	2: (* === Check loop *)
		IF NOT (MB_Lock OR MB_Start) THEN
			WHILE VarCnt<=(VARS_Max-1) AND VarSta=2 DO
				(* Check only active vars *)
				IF VARS[VarCnt].Variable<>0 THEN			(* "Variable" is a pointer to word, so if 0 no address *)
					(* Check var auto-refresh on timer checks *)
					IF VARS[VarCnt].Refresh_Time>0 AND VARS[VarCnt].Refresh_Cnt=0 THEN
						VARS[VarCnt].Refresh_Cnt:=VARS[VarCnt].Refresh_Time;
						VarSta:=3;
					END_IF
					(* Check refresh for change or request *)
					CASE VARS[VarCnt].FunCode OF
						5,6,15,16: (* Write functions *)
							IF VARS[VarCnt].Variable_Size=1 THEN
								IF VARS[VarCnt].Variable^<>VARS[VarCnt].Variable_Mirror THEN
									VARS[VarCnt].Variable_Mirror:=VARS[VarCnt].Variable^;
									VarSta:=3;
								END_IF
							ELSE
								IF VARS[VarCnt].Variable_Mirror<>0 THEN
									VARS[VarCnt].Variable_Mirror:=0;
									VarSta:=3;
								END_IF
							END_IF
						1,2,3,4: (* Read functions *)
							IF VARS[VarCnt].Variable_Mirror<>0 THEN
								VARS[VarCnt].Variable_Mirror:=0;
								VarSta:=3;
							END_IF
					END_CASE
				END_IF
				(* Process query *)
				IF VarSta=3 THEN
					MB_Lock:=TRUE;
					MB_Query.SlaveAddress:=VARS[VarCnt].SlaveAddress;
					MB_Query.FunctionCode:=VARS[VarCnt].FunCode;
					CASE VARS[VarCnt].FunCode OF
						16#5,16#6,16#F,16#10:
							MB_Query.Read_Quantity:=0;
							MB_Query.Read_StartAddress:=0;
							MB_Query.Write_StartAddress:=VARS[VarCnt].FunAddress;
							MB_Query.Write_Quantity:=VARS[VarCnt].Variable_Size;
							IF VARS[VarCnt].Variable_Size=200 THEN
								COPY_32SWAP16(VARS[VarCnt].Variable, ADR(MB_Query.Write_Data[0]));
							ELSIF VARS[VarCnt].Variable_Size>1 THEN
								MEMCPY(VARS[VarCnt].Variable, ADR(MB_Query.Write_Data[0]), 2*VARS[VarCnt].Variable_Size);
							ELSE
								MB_Query.Write_Data[0]:=VARS[VarCnt].Variable^;
							END_IF
						16#1,16#2,16#3,16#4:
							MB_Query.Read_StartAddress:=VARS[VarCnt].FunAddress;
							IF VARS[VarCnt].Variable_Size=200 THEN MB_Query.Read_Quantity:=2; ELSE
							  MB_Query.Read_Quantity:=VARS[VarCnt].Variable_Size;
							END_IF
							MB_Query.Write_StartAddress:=0;
							MB_Query.Write_Quantity:=0;
					END_CASE
					VarRetry:=0;
					MB_Start:=TRUE;
				ELSE
					VarCnt:=VarCnt+1;
				END_IF
			END_WHILE
			(* Check loop completed -> no actions *)
			IF VarSta=2 THEN VarSta:=1; END_IF
		END_IF

	3: (* === Wait & process MB response *)
		IF NOT MB_Start THEN
			IF MB_MASTER.MB_Error=0 THEN
				CASE VARS[VarCnt].FunCode OF
					1,2,3,4:
						IF VARS[VarCnt].Variable_Size=200 THEN
							COPY_32SWAP16(ADR(MB_Resp.Data), VARS[VarCnt].Variable);
						ELSIF VARS[VarCnt].Variable_Size>1 THEN
							MEMCPY(ADR(MB_Resp.Data), VARS[VarCnt].Variable, 2*VARS[VarCnt].Variable_Size);
						ELSE
							VARS[VarCnt].Variable^:=MB_Resp.Data[0];
						END_IF
				END_CASE
				MB_Lock:=FALSE;
				(* Signal error recovery *)
				IF VARS_Alarm=TRUE AND VarCnt=VarAlarm THEN
					LogEv(EL_Wrn,EO_MODBUS,ID,5,'');
					VARS_Alarm:=FALSE;
				END_IF
				(* Next var *)
				VarCnt:=VarCnt+1;
				VarSta:=2;
			ELSE
				IF VarRetry<3 THEN
					VarRetry:=VarRetry+1;
					MB_Start:=TRUE;
				ELSE
					MB_Lock:=FALSE;
					(* Signal error *)
					IF VARS_Alarm=FALSE THEN
						LogEv(EL_Wrn,EO_MODBUS,ID,3,INT_TO_STRING(MB_MASTER.MB_Error));
						VARS_Alarm:=TRUE;
						VarAlarm:=VarCnt-1;
					END_IF
					(* Next var *)
					VarCnt:=VarCnt+1;
					VarSta:=2;
				END_IF
			END_IF
		END_IF

ELSE
	VarSta:=0;
END_CASE
END_ACTION

(* POU Plant_Objects/obj_MODBUS_CIR, ST *)
FUNCTION_BLOCK obj_MODBUS_CIR
VAR CONSTANT
	WAIT_STATE		:	BYTE := 0;
	PUMP_STATUS		:	BYTE := 1;
	PUMP_DATA		:	BYTE := 2;
	PUMP_ALARMS		:	BYTE := 3;
	PUMP_END_READ	:	BYTE := 4;
	CIR_ON_OFF		:	BYTE := 90;
	CIR_ON_OFF_CHECK:	BYTE := 91;
	CIR_END_WRITE	:	BYTE := 92;
	ERROR_STATE		:	BYTE := 100;
END_VAR
VAR_INPUT
	ID		:	BYTE;
	Address :	BYTE;		(* Pump address *)

	(* Physical inputs *)
	CIR_RUN_REQ		: BOOL; (* External run request (no heat or cold requested) *)
	CIR_STOP_REQ	: BOOL; (* External stop request (has priority over RUN signals!) *)

	Pump_AL			: BOOL; (* Alarm input signal *)
	Pump_AUTO		: BOOL;	(* Automatic/Manual input *)

	(* Controls *)
	OnOff		: 	BOOL;
	InitOK		:	BOOL;

	(* Timings *)
	OnDelay		:	TIME;
	OffDelay	:	TIME;

	(* Modbus *)
	Refresh_Now	:	BOOL;	(* Start immediately modbus state machine *)
END_VAR
VAR_IN_OUT
	ModBus		:	obj_MODBUS;
END_VAR
VAR_OUTPUT
	Ctrl_Run	:	BOOL;		(* Logical status of the device: 0: Not running (switched off), 1: running *)
	Run			:	BOOL;		(* Real status *)

	Status_Log	:	WORD;
	Status_Vis	:	DWORD;
END_VAR
VAR
	Pump_En		:	BOOL;

	(* Filters *)
	fPump_AL	:	FLT_EVENT := (INITEV:=FALSE);
	fPump_ST	:	FLT_EVENT := (INITEV:=FALSE);
	fPump_En	:	FLT_EVENT;
	fCIR_AUTO	:	FLT_EVENT;
	fStatus		:	FLT_EVENT;
	fStatusFault:	BOOL;

	(* Timer manage switch on/off delay *)
	Delay		: 	TONOF;

	(* CIR data structure *)
	DataPump	:	typ_MODBUS_CIR;

	(* Modbus variables *)
	state		:	BYTE;
	retry		:	BYTE;
	ReadTmr		:	TON := (PT:=T#5m);
	fModbusAlr	: 	BOOL;
	fWrite		:	BOOL;

	(* Alarm and Warning counters *)
	AlarmCtr	:	BYTE;
	WarningCtr	:	BYTE;

	(* Filers on alarms and faults *)
	AlarmHw		:	FLT_EVENT := (INITEV:=FALSE);
	Alarm		:	FLT_EVENT := (INITEV:=FALSE);
	Inverter	:	FLT_EVENT := (INITEV:=FALSE);
	ModbusAlr	:	FLT_EVENT := (INITEV:=FALSE);

	OldAlarm	:	WORD;

END_VAR
Init();

PumpManager();

(* State machine to read pump parameters *)
Stm();

(* Check alarm and warning for both pumps *)
CheckFault();

(* Set output according to logical On/Off status *)
IF AlarmCtr>0 THEN Run := FALSE;
ELSE Run := Ctrl_Run;
END_IF

IF AlarmCtr>0 THEN
	Status_Log := 2;
	Status_Vis := COLOR_RED;
ELSIF WarningCtr>0 THEN
	Status_Log := 1;
	Status_Vis := COLOR_YELLOW;
ELSE
	Status_Log := 0;
	Status_Vis := COLOR_GREEN;
END_IF

(* Update error lamp status *)
Lamp.UpdateStatus(obj_Status:=Status_Log);
END_FUNCTION_BLOCK
ACTION AddLogData:
Logger.s1:=INSERT('&CIR=',BYTE_TO_STRING(ID),4);
IF ID<10 THEN Logger.s1:=INSERT(Logger.s1,'0',4); END_IF

Logger.s1:=CONCAT(Logger.s1,WORD_TO_STRING(DataPump.PumpStatus));		Logger.s1:=CONCAT(Logger.s1,';');
Logger.s1:=CONCAT(Logger.s1,INT_TO_STRING(DataPump.PumpBoardTemp));		Logger.s1:=CONCAT(Logger.s1,';');
Logger.s1:=CONCAT(Logger.s1,WORD_TO_STRING(DataPump.PumpVoltage));		Logger.s1:=CONCAT(Logger.s1,';');
Logger.s1:=CONCAT(Logger.s1,WORD_TO_STRING(DataPump.PumpRPM));			Logger.s1:=CONCAT(Logger.s1,';');
Logger.s1:=CONCAT(Logger.s1,WORD_TO_STRING(DataPump.PumpPower));		Logger.s1:=CONCAT(Logger.s1,';');
Logger.s1:=CONCAT(Logger.s1,DWORD_TO_STRING(DataPump.PumpOpTime));		Logger.s1:=CONCAT(Logger.s1,';');
Logger.s1:=CONCAT(Logger.s1,WORD_TO_STRING(DataPump.PumpHead));			Logger.s1:=CONCAT(Logger.s1,';');
Logger.s1:=CONCAT(Logger.s1,WORD_TO_STRING(DataPump.PumpFlow));			Logger.s1:=CONCAT(Logger.s1,';');
Logger.s1:=CONCAT(Logger.s1,WORD_TO_STRING(DataPump.PumpLiqTemp));		Logger.s1:=CONCAT(Logger.s1,';');

Logger.s1:=CONCAT(Logger.s1,WORD_TO_STRING(Status_Log));
ADDSTRING(ADR(Logger.TData), ADR(Logger.s1), Logger.TLen);
END_ACTION
ACTION CheckFault:
(*** WARNINGS ***)

(* Verify ModBus error	*)
ModbusAlr(IN:=fModbusAlr);

IF ModbusAlr.EVH THEN
	LogEv(EL_Wrn,EO_CIR,ID,13,SEL(ModBus.MB_MASTER.MB_Error<>0,'0','1'));
	WarningCtr := 1;
END_IF

IF ModbusAlr.EVL THEN WarningCtr := 0; END_IF



(*** ALARMS ***)

(* Hardware alarm (physical input *)
AlarmHw(IN:=Pump_AL);

IF AlarmHw.EVH THEN
	LogEv(EL_Alarm,EO_CIR,ID,3,'CIR_Alarm');
	AlarmCtr := AlarmCtr + 1;
END_IF

IF AlarmHw.EVL THEN
	LogEv(EL_Log,EO_CIR,ID,4,'CIR_Alarm_Recovered');
	AlarmCtr := AlarmCtr - 1;
END_IF

(* General alarm (read by Modbus) *)
Alarm(IN:=(DataPump.PumpAlarm[0] <> OldAlarm));

IF Alarm.EVH THEN
	IF DataPump.PumpAlarm[0] = 0 THEN
		LogEv(EL_Log,EO_CIR,ID,12,'Alarm_Recovered');
		AlarmCtr := AlarmCtr - 1;
	ELSE
		LogEv(EL_Alarm,EO_CIR,ID,11,WORD_TO_STRING(DataPump.PumpAlarm[0]));
		AlarmCtr := AlarmCtr + 1;
	END_IF

	OldAlarm := DataPump.PumpAlarm[0];
END_IF

(* Inverter pump error *)
Inverter(IN:=DataPump.PumpFault);

IF Inverter.EVH THEN
	LogEv(EL_Alarm,EO_CIR,ID,9,'Inverter_Fault');
	AlarmCtr := AlarmCtr + 1;
END_IF

IF Inverter.EVL THEN
	LogEv(EL_Alarm,EO_CIR,ID,10,'Inverter_Fault_Recovered');
	AlarmCtr := AlarmCtr - 1;
END_IF
END_ACTION
ACTION Init:
IF NOT InitOK THEN

	Delay.PT_OF := SEL(OffDelay=T#0s, OffDelay, Plant_CirOffDelay);
	Delay.PT_ON := SEL(OffDelay=T#0s, OnDelay, Plant_CirOnDelay) + WORD_TO_TIME(1000*ID);

	InitOK := TRUE;

END_IF
END_ACTION
ACTION PumpManager:
(*** Verify Status ***)
IF (Pump_En AND DataPump.PumpStatus=0) OR (NOT Pump_En AND DataPump.PumpStatus=2) THEN fStatusFault := TRUE;
ELSE fStatusFault := FALSE;
END_IF

fPump_ST(IN:=fStatusFault);

IF fPump_ST.EVH THEN
	LogEv(SEL(Pump_En,EL_Alarm,EL_Wrn),EO_CIRD,ID,SEL(Pump_En,5,6),'');
	WarningCtr := WarningCtr + 1;
END_IF

IF fPump_ST.EVL THEN WarningCtr := WarningCtr - 1; END_IF

(* Verify if in Auto or Manual mode *)
fCIR_AUTO(IN:=Pump_AUTO);

(* MANUAL MODE *)
IF fCIR_AUTO.EVH THEN
	LogEv(EL_Log,EO_CIR,ID,8,'CIR_Auto');
	WarningCtr := WarningCtr - 1;
END_IF

(* Manual -> Keep switched on *)
IF fCIR_AUTO.EVL THEN
	LogEv(EL_Wrn,EO_CIR,ID,7,'CIR_Manual');
	WarningCtr := WarningCtr + 1;
END_IF

(* Verify if OnOff is changed *)
fStatus(IN:=OnOff);

IF fStatus.EVH THEN Ctrl_Run := TRUE; END_IF
IF fStatus.EVL THEN Ctrl_Run := FALSE; END_IF

(* Check switch on or switch off delay *)
Delay(IN:=Ctrl_Run);

IF Pump_AUTO THEN
	(* If priority request *)
	IF CIR_STOP_REQ THEN Pump_En := 1;
	ELSIF CIR_RUN_REQ THEN Pump_En := 0;
	ELSE Pump_En := NOT Delay.OUT;
	END_IF
	
	(* Set RUN signal (for external objects) *)
	IF fPump_AL.IN OR fPump_ST.IN THEN
		Ctrl_Run:=FALSE;
	ELSE
		Run:=Delay.OUT;
	END_IF
END_IF

(* Check if a pump enable update (modbus write) is requested *)
fPump_En(IN:=Pump_En);

IF fPump_En.EVH OR fPump_En.EVL THEN
	fWrite := TRUE;
	Refresh_Now := TRUE;
END_IF
END_ACTION
ACTION Stm:
CASE state OF
	WAIT_STATE:	(* Refresh time manager *)
		ReadTmr(IN:=NOT ReadTmr.Q);
		IF ReadTmr.Q OR Refresh_Now  THEN
			state := PUMP_STATUS;
			ReadTmr.PT := T#1m;
			Refresh_Now := FALSE;
		END_IF

	(**** READ CIR PARAMETERS ****)

	PUMP_STATUS:	(* Status and Fault *)
		Modbus.MB_Lock := TRUE;
		Modbus.MB_Query.SlaveAddress := Address;
		Modbus.MB_Query.FunctionCode := 3;
		ModBus.MB_Query.Read_StartAddress := 201;
		ModBus.MB_Query.Read_Quantity := 2;
		ModBus.MB_Start := TRUE;

		state := PUMP_DATA;

	PUMP_DATA:	(* Pump data *)
		IF NOT ModBus.MB_Start THEN
			IF ModBus.MB_MASTER.bInterfaceError<>0 OR ModBus.MB_MASTER.MB_Error<>0 THEN
				state := ERROR_STATE;
			ELSE
				DataPump.PumpStatus := ModBus.MB_Resp.Data[0];
				DataPump.PumpFault	:= WORD_TO_BOOL(ModBus.MB_Resp.Data[1]);

				ModBus.MB_Query.Read_StartAddress := 210;
				ModBus.MB_Query.Read_Quantity := 12;
				ModBus.MB_Start := TRUE;

				state := PUMP_ALARMS;
			END_IF
		END_IF

	PUMP_ALARMS: (* Historical alarms *)
		IF NOT ModBus.MB_Start THEN
			IF ModBus.MB_MASTER.bInterfaceError<>0 OR ModBus.MB_MASTER.MB_Error<>0 THEN
				state := ERROR_STATE;
			ELSE
				DataPump.PumpBoardTemp 	:= WORD_TO_INT(ModBus.MB_Resp.Data[0]);
				DataPump.PumpVoltage	:= ModBus.MB_Resp.Data[2];
				DataPump.PumpCurrent	:= ModBus.MB_Resp.Data[3];
				DataPump.PumpRPM		:= ModBus.MB_Resp.Data[5];
				DataPump.PumpPower		:= ModBus.MB_Resp.Data[6];
				DataPump.PumpOpTime		:= BUILD_16TO32(ADR(ModBus.MB_Resp.Data[7]));
				DataPump.PumpHead		:= ModBus.MB_Resp.Data[9];
				DataPump.PumpFlow		:= ModBus.MB_Resp.Data[10];
				DataPump.PumpLiqTemp	:= WORD_TO_INT(ModBus.MB_Resp.Data[11]);


				ModBus.MB_Query.Read_StartAddress := 230;
				ModBus.MB_Query.Read_Quantity := 15;
				ModBus.MB_Start := TRUE;

				state := PUMP_END_READ;
			END_IF
		END_IF

	PUMP_END_READ:	(* Read alarms *)
		IF NOT ModBus.MB_Start THEN
			IF ModBus.MB_MASTER.bInterfaceError<>0 OR ModBus.MB_MASTER.MB_Error<>0 THEN
				state := ERROR_STATE;
			ELSE
				DataPump.PumpAlarm[0] := ModBus.MB_Resp.Data[0];
				DataPump.PumpAlarm[1] := ModBus.MB_Resp.Data[1];
				DataPump.PumpAlarm[2] := ModBus.MB_Resp.Data[2];
				DataPump.PumpAlarm[3] := ModBus.MB_Resp.Data[3];
				DataPump.PumpAlarm[4] := ModBus.MB_Resp.Data[4];
				DataPump.PumpAlarm[5] := ModBus.MB_Resp.Data[5];
				DataPump.PumpAlarm[6] := ModBus.MB_Resp.Data[6];
				DataPump.PumpAlarm[7] := ModBus.MB_Resp.Data[7];
				DataPump.PumpAlarm[8] := ModBus.MB_Resp.Data[8];
				DataPump.PumpAlarm[9] := ModBus.MB_Resp.Data[9];
				DataPump.PumpAlarm[10] := ModBus.MB_Resp.Data[10];
				DataPump.PumpAlarm[11] := ModBus.MB_Resp.Data[11];
				DataPump.PumpAlarm[12] := ModBus.MB_Resp.Data[12];
				DataPump.PumpAlarm[13] := ModBus.MB_Resp.Data[13];
				DataPump.PumpAlarm[14] := ModBus.MB_Resp.Data[14];

				IF fModbusAlr THEN fModbusAlr := FALSE; END_IF

				IF fWrite THEN state := CIR_ON_OFF;
				ELSE
					ModBus.MB_Lock := FALSE;
					retry := 0;
					state := WAIT_STATE;
				END_IF
			END_IF
		END_IF

	(**** WRITE ON/OFF REGISTER AND VERIFY RIGHT SETTING ****)
	CIR_ON_OFF:	(* Pump On/off *)

		Modbus.MB_Query.SlaveAddress := Address;
		Modbus.MB_Query.FunctionCode := 6;
		ModBus.MB_Query.Write_StartAddress := 110;
		ModBus.MB_Query.Write_Quantity := 1;
		ModBus.MB_Query.Write_Data[0] := BOOL_TO_WORD(OnOff);
		ModBus.MB_Start := TRUE;

		state := CIR_END_WRITE;

	CIR_END_WRITE:
		IF NOT ModBus.MB_Start THEN
			IF ModBus.MB_MASTER.bInterfaceError<>0 OR ModBus.MB_MASTER.MB_Error<>0 THEN
				state := ERROR_STATE;
			ELSE
				fWrite := FALSE;

				ModBus.MB_Lock := FALSE;
				retry := 0;
				state := WAIT_STATE;
				fWrite := FALSE;
			END_IF
		END_IF


	(**** CHECK MODBUS ERROR ****)
	ERROR_STATE: 	(* Release MODBUS *)
			MODBUS.MB_Lock:=FALSE;

			(* Retries *)
			retry:=retry+1;
			IF retry>3 THEN
				retry:=0;
				(* Signal event *)
				fModbusAlr := TRUE;
			END_IF

			state:=WAIT_STATE;
END_CASE
END_ACTION

(* POU Plant_Objects/obj_MODBUS_CIR_DOPPIO, ST *)
FUNCTION_BLOCK obj_MODBUS_CIR_DOPPIO
VAR CONSTANT
	WAIT_STATE		:	BYTE := 0;
	PUMP1_STATUS	:	BYTE := 1;
	PUMP1_DATA		:	BYTE := 2;
	PUMP1_ALARMS	:	BYTE := 3;
	PUMP1_END_READ	:	BYTE := 4;
	PUMP2_STATUS	:	BYTE := 5;
	PUMP2_DATA		:	BYTE := 6;
	PUMP2_ALARMS	:	BYTE := 7;
	PUMP2_END_READ	:	BYTE := 8;
	CIR_ON_OFF		:	BYTE := 90;
	CIR_ON_OFF_CHECK:	BYTE := 91;
	CIR_END_WRITE	:	BYTE := 92;
	ERROR_STATE		:	BYTE := 100;
END_VAR
VAR_INPUT
	ID		:	BYTE;
	Address1:	BYTE;		(* Pump 1 address *)
	Address2:	BYTE;		(* Pump 2 address *)

	(* Controls *)
	Ctrl_SetPoint 	: INT;
	CIR_RUN_REQ		: BOOL; (* External run request (no heat or cold requested) *)
	CIR_STOP_REQ	: BOOL; (* External stop request (has priority over RUN signals!) *)

	PumpA_AL		: BOOL; (* Alarm input signal *)
	PumpB_AL		: BOOL;

	PumpA_AUTO		: BOOL;
	PumpB_AUTO		: BOOL;

	OnOff			: BYTE;
END_VAR
VAR_IN_OUT
	ModBus		:	obj_MODBUS;
END_VAR
VAR_OUTPUT
	Run			:	BOOL;

	Status_Log	:	WORD;
	Status_Vis	:	DWORD;
END_VAR
VAR
	Ctrl_Run	:	BOOL;		(* Logical status of the device: 0: Not running (switched off), 1: running *)
	CIR_AUTO	:	BOOL;
	CirStatus	:	BYTE;
	OldCirStatus:	BYTE;
	fWrite		:	BOOL;

	state		:	BYTE;
	retry		:	BYTE;
	ReadTmr		:	TON := (PT:=T#5m);
	retry_write	:	BYTE;

	DataPump1	:	typ_MODBUS_CIR;
	DataPump2	:	typ_MODBUS_CIR;

	OldAlarmPump1	:	WORD;
	OldAlarmPump2	:	WORD;

	fWrn1		:	BOOL;
	fWrn2		:	BOOL;

	fStatus		:	FLT_EVENT;
	fCIR_AUTO	:	FLT_EVENT;
	Alarm1		:	FLT_EVENT;
	Alarm2		:	FLT_EVENT;
	AlarmHw1	:	FLT_EVENT := (INITEV:=FALSE);
	AlarmHw2	:	FLT_EVENT := (INITEV:=FALSE);
	Inverter1	:	FLT_EVENT := (INITEV:=FALSE);
	Inverter2	:	FLT_EVENT := (INITEV:=FALSE);
	Warning1	:	FLT_EVENT := (INITEV:=FALSE);
	Warning2	:	FLT_EVENT := (INITEV:=FALSE);

	s1			:	STRING;
	Delay		: 	TONOF := (PT_OF:=Plant_CirOffDelay);
END_VAR
ManagePump();

(* State machine to read pump parameters *)
Stm();

(* Check alarm and warning for both pumps *)
CheckFault();

IF Status_Log = 2 THEN Run := FALSE;
ELSE Run := Ctrl_Run;
END_IF

Lamp.obj_Status := Status_Log;
Lamp.UpdateStatus();

IF Status_Log = 2 THEN Status_Vis := COLOR_RED;
ELSIF Status_Log = 1 THEN Status_Vis := COLOR_YELLOW;
ELSE Status_Vis := COLOR_GREEN;
END_IF
END_FUNCTION_BLOCK
ACTION AddLogData:
Logger.s1:=INSERT('&CIR=',BYTE_TO_STRING(ID),4);
IF ID<10 THEN Logger.s1:=INSERT(Logger.s1,'0',4); END_IF

(* PUMP 1 *)
Logger.s1:=CONCAT(Logger.s1,WORD_TO_STRING(DataPump1.PumpStatus));		Logger.s1:=CONCAT(Logger.s1,';');
Logger.s1:=CONCAT(Logger.s1,INT_TO_STRING(DataPump1.PumpBoardTemp));	Logger.s1:=CONCAT(Logger.s1,';');
Logger.s1:=CONCAT(Logger.s1,WORD_TO_STRING(DataPump1.PumpVoltage));		Logger.s1:=CONCAT(Logger.s1,';');
Logger.s1:=CONCAT(Logger.s1,WORD_TO_STRING(DataPump1.PumpRPM));			Logger.s1:=CONCAT(Logger.s1,';');
Logger.s1:=CONCAT(Logger.s1,WORD_TO_STRING(DataPump1.PumpPower));		Logger.s1:=CONCAT(Logger.s1,';');
Logger.s1:=CONCAT(Logger.s1,DWORD_TO_STRING(DataPump1.PumpOpTime));		Logger.s1:=CONCAT(Logger.s1,';');
Logger.s1:=CONCAT(Logger.s1,WORD_TO_STRING(DataPump1.PumpHead));		Logger.s1:=CONCAT(Logger.s1,';');
Logger.s1:=CONCAT(Logger.s1,WORD_TO_STRING(DataPump1.PumpFlow));		Logger.s1:=CONCAT(Logger.s1,';');
Logger.s1:=CONCAT(Logger.s1,WORD_TO_STRING(DataPump1.PumpLiqTemp));		Logger.s1:=CONCAT(Logger.s1,';');

(* PUMP 2 *)
Logger.s1:=CONCAT(Logger.s1,WORD_TO_STRING(DataPump2.PumpStatus));		Logger.s1:=CONCAT(Logger.s1,';');
Logger.s1:=CONCAT(Logger.s1,INT_TO_STRING(DataPump2.PumpBoardTemp));	Logger.s1:=CONCAT(Logger.s1,';');
Logger.s1:=CONCAT(Logger.s1,WORD_TO_STRING(DataPump2.PumpVoltage));		Logger.s1:=CONCAT(Logger.s1,';');
Logger.s1:=CONCAT(Logger.s1,WORD_TO_STRING(DataPump2.PumpRPM));			Logger.s1:=CONCAT(Logger.s1,';');
Logger.s1:=CONCAT(Logger.s1,WORD_TO_STRING(DataPump2.PumpPower));		Logger.s1:=CONCAT(Logger.s1,';');
Logger.s1:=CONCAT(Logger.s1,DWORD_TO_STRING(DataPump2.PumpOpTime));		Logger.s1:=CONCAT(Logger.s1,';');
Logger.s1:=CONCAT(Logger.s1,WORD_TO_STRING(DataPump2.PumpHead));		Logger.s1:=CONCAT(Logger.s1,';');
Logger.s1:=CONCAT(Logger.s1,WORD_TO_STRING(DataPump2.PumpFlow));		Logger.s1:=CONCAT(Logger.s1,';');
Logger.s1:=CONCAT(Logger.s1,WORD_TO_STRING(DataPump2.PumpLiqTemp));		Logger.s1:=CONCAT(Logger.s1,';');

Logger.s1:=CONCAT(Logger.s1,WORD_TO_STRING(Status_Log));
ADDSTRING(ADR(Logger.TData), ADR(Logger.s1), Logger.TLen);
END_ACTION
ACTION CheckFault:
(**** PUMP 1 ****)
AlarmHw1(IN:=PumpA_AL);

IF AlarmHw1.EVH THEN
	LogEv(EL_Alarm,EO_CIRD,ID,3,'CIR_Alarm_A');
	Status_Log := 2;
END_IF

IF AlarmHw1.EVL THEN
	LogEv(EL_Alarm,EO_CIRD,ID,4,'CIR_Alarm_A_Recovered');
	Status_Log := 0;
END_IF

Inverter1(IN:=DataPump1.PumpFault);

IF Inverter1.EVH THEN
	LogEv(EL_Alarm,EO_CIRD,ID,15,'Inverter_Fault_A');
	Status_Log := 2;
END_IF

IF Inverter1.EVL THEN
	LogEv(EL_Alarm,EO_CIRD,ID,16,'Inverter_Fault_A_Recovered');
	Status_Log := 0;
END_IF

Alarm1(IN:=(DataPump1.PumpAlarm[0] <> OldAlarmPump1));

IF Alarm1.EVH THEN
	IF DataPump1.PumpAlarm[0] = 0 THEN
		LogEv(EL_Alarm,EO_CIRD,ID,18,'Alarm_A_Recovered');
		Status_Log := 0;
	ELSE
		s1 := WORD_TO_STRING(DataPump1.PumpAlarm[0]);
		LogEv(EL_Alarm,EO_CIRD,ID,17,s1);
		Status_Log := 2;
	END_IF

	OldAlarmPump1 := DataPump1.PumpAlarm[0];
END_IF

IF DataPump1.PumpLiqTemp < 5 OR DataPump1.PumpLiqTemp > 80 THEN fWrn1 := TRUE;
ELSE fWrn1 := FALSE;
END_IF

Warning1(IN:=fWrn1);

IF Warning1.EVH THEN
	LogEv(EL_Wrn,EO_CIRD,ID,19,'Liquid_Temperature_A');

	IF Status_Log <> 2 THEN Status_Log := 1; END_IF
END_IF

IF Warning1.EVL THEN
	LogEv(EL_Log,EO_CIRD,ID,20,'Liquid_Temperature_A_Recovered');
	Status_Log := 0;
END_IF

(**** PUMP 2 ****)
AlarmHw2(IN:=PumpB_AL);

IF AlarmHw2.EVH THEN
	LogEv(EL_Alarm,EO_CIRD,ID,11,'CIR_Alarm_B');
	Status_Log := 2;
END_IF

IF AlarmHw2.EVL THEN
	LogEv(EL_Alarm,EO_CIRD,ID,12,'CIR_Alarm_B_Recovered');
	Status_Log := 0;
END_IF

Inverter2(IN:=DataPump2.PumpFault);

IF Inverter2.EVH THEN
	LogEv(EL_Alarm,EO_CIRD,ID,21,'Inverter_Fault_B');
	Status_Log := 2;
END_IF

IF Inverter2.EVL THEN
	LogEv(EL_Alarm,EO_CIRD,ID,22,'Inverter_Fault_B_Recovered');
	Status_Log := 0;
END_IF

Alarm2(IN:=(DataPump2.PumpAlarm[0] <> OldAlarmPump2));

IF Alarm2.EVH THEN
	IF DataPump2.PumpAlarm[0] = 0 THEN
		LogEv(EL_Log,EO_CIRD,ID,24,'Alarm_B_Recovered');
		Status_Log := 0;
	ELSE
		s1 := WORD_TO_STRING(DataPump2.PumpAlarm[0]);
		LogEv(EL_Alarm,EO_CIRD,ID,23,s1);
		Status_Log := 2;
	END_IF

	OldAlarmPump2 := DataPump2.PumpAlarm[0];
END_IF

IF DataPump2.PumpLiqTemp < 5 OR DataPump2.PumpLiqTemp > 80 THEN fWrn2 := TRUE;
ELSE fWrn2 := FALSE;
END_IF

Warning2(IN:=fWrn2);

IF Warning2.EVH THEN
	LogEv(EL_Wrn,EO_CIRD,ID,25,'Liquid_Temperature_B');

	IF Status_Log <> 2 THEN Status_Log := 1; END_IF
END_IF

IF Warning2.EVL THEN
	LogEv(EL_Log,EO_CIRD,ID,26,'Liquid_Temperature_B_Recovered');
	Status_Log := 0;
END_IF

(*
IF Status_Log = 0 THEN
	LogEv(EL_Log,0,ID,1,'');
END_IF*)
END_ACTION
ACTION ManagePump:
CIR_AUTO := PumpA_AUTO OR PumpB_AUTO;

OldCirStatus := CirStatus;

fCIR_AUTO(IN:=CIR_AUTO);
IF fCIR_AUTO.EVL THEN
	LogEv(EL_Wrn,EO_CIRD,ID,7,'CIR_Manual');

	(* MANUAL MODE	-> CIR working depends on external signal *)
	CirStatus := 2;
	fWrite := TRUE;

END_IF

IF fCIR_AUTO.EVH THEN LogEv(EL_Log,EO_CIRD,ID,8,'CIR_Auto'  ); END_IF

(* AUTOMATIC MODE *)
IF CIR_AUTO THEN

	IF OnOff = 0 THEN
	
		Ctrl_Run := FALSE;			(* Logically swtched off *)
		Delay(IN:=Ctrl_Run);		(* Count delay time before physical switch off	*)

	ELSIF OnOff = 1 THEN

		(* Start switch on delay time (proportional to object id) *)
		Delay(IN:=TRUE, PT_ON:=WORD_TO_TIME(1000*ID));
	
		IF NOT Ctrl_Run AND Delay.OUT THEN
			Ctrl_Run := TRUE;				(* Set logical running variable as true -> CIR running *)
		END_IF
	
	ELSE
		Delay(IN:=TRUE, PT_ON:=T#0s);		(* Antifreeze -> Enable immediatly *)
	END_IF
	
	IF CIR_STOP_REQ    THEN CirStatus:=0;
	ELSIF CIR_RUN_REQ  THEN CirStatus:=1;
					   ELSE CirStatus:=BOOL_TO_BYTE(Delay.OUT); END_IF
	
	(* If functioning status has changed, phisically modify it according to variable state, otherwise keep same status *)
	fStatus(IN:=(CirStatus <> OldCirStatus));

	IF fStatus.EVH THEN
		fWrite := TRUE;
	END_IF

END_IF
END_ACTION
ACTION Stm:
CASE state OF
	WAIT_STATE:	(* Refresh time manager *)
		ReadTmr(IN:=NOT ReadTmr.Q);
		IF ReadTmr.Q THEN
			state := PUMP1_STATUS;
			ReadTmr.PT := T#60s;
		END_IF

		IF fWrite THEN
			state := CIR_ON_OFF;
			fWrite := FALSE;
		END_IF

	(**** READ CIR PARAMETERS ****)

	(**** PUMP 1 ****)
	PUMP1_STATUS:	(* Status and Fault *)
		Modbus.MB_Lock := TRUE;
		Modbus.MB_Query.SlaveAddress := Address1;
		Modbus.MB_Query.FunctionCode := 3;
		ModBus.MB_Query.Read_StartAddress := 201;
		ModBus.MB_Query.Read_Quantity := 2;
		ModBus.MB_Start := TRUE;

		state := PUMP1_DATA;

	PUMP1_DATA:	(* Pump data *)
		IF NOT ModBus.MB_Start THEN
			IF ModBus.MB_MASTER.bInterfaceError<>0 THEN
				state := ERROR_STATE;
			ELSE
				DataPump1.PumpStatus := ModBus.MB_Resp.Data[0];
				DataPump1.PumpFault	:= WORD_TO_BOOL(ModBus.MB_Resp.Data[1]);

				ModBus.MB_Query.Read_StartAddress := 210;
				ModBus.MB_Query.Read_Quantity := 12;
				ModBus.MB_Start := TRUE;

				state := PUMP1_ALARMS;
			END_IF
		END_IF

	PUMP1_ALARMS: (* Historical alarms *)
		IF NOT ModBus.MB_Start THEN
			IF ModBus.MB_MASTER.bInterfaceError<>0 THEN
				state := ERROR_STATE;
			ELSE
				DataPump1.PumpBoardTemp := WORD_TO_INT(ModBus.MB_Resp.Data[0]);
				DataPump1.PumpVoltage	:= ModBus.MB_Resp.Data[2];
				DataPump1.PumpCurrent	:= ModBus.MB_Resp.Data[3];
				DataPump1.PumpRPM		:= ModBus.MB_Resp.Data[5];
				DataPump1.PumpPower		:= ModBus.MB_Resp.Data[6];
				DataPump1.PumpOpTime	:= BUILD_16TO32(ADR(ModBus.MB_Resp.Data[7]));
				DataPump1.PumpHead		:= ModBus.MB_Resp.Data[9];
				DataPump1.PumpFlow		:= ModBus.MB_Resp.Data[10];
				DataPump1.PumpLiqTemp	:= WORD_TO_INT(ModBus.MB_Resp.Data[11]);


				ModBus.MB_Query.Read_StartAddress := 230;
				ModBus.MB_Query.Read_Quantity := 15;
				ModBus.MB_Start := TRUE;

				state := PUMP1_END_READ;
			END_IF
		END_IF

	PUMP1_END_READ:	(* Read alarms *)
		IF NOT ModBus.MB_Start THEN
			IF ModBus.MB_MASTER.bInterfaceError<>0 THEN
				state := ERROR_STATE;
			ELSE
				DataPump1.PumpAlarm[0] := ModBus.MB_Resp.Data[0];
				DataPump1.PumpAlarm[1] := ModBus.MB_Resp.Data[1];
				DataPump1.PumpAlarm[2] := ModBus.MB_Resp.Data[2];
				DataPump1.PumpAlarm[3] := ModBus.MB_Resp.Data[3];
				DataPump1.PumpAlarm[4] := ModBus.MB_Resp.Data[4];
				DataPump1.PumpAlarm[5] := ModBus.MB_Resp.Data[5];
				DataPump1.PumpAlarm[6] := ModBus.MB_Resp.Data[6];
				DataPump1.PumpAlarm[7] := ModBus.MB_Resp.Data[7];
				DataPump1.PumpAlarm[8] := ModBus.MB_Resp.Data[8];
				DataPump1.PumpAlarm[9] := ModBus.MB_Resp.Data[9];
				DataPump1.PumpAlarm[10] := ModBus.MB_Resp.Data[10];
				DataPump1.PumpAlarm[11] := ModBus.MB_Resp.Data[11];
				DataPump1.PumpAlarm[12] := ModBus.MB_Resp.Data[12];
				DataPump1.PumpAlarm[13] := ModBus.MB_Resp.Data[13];
				DataPump1.PumpAlarm[14] := ModBus.MB_Resp.Data[14];

				state := PUMP2_STATUS;
			END_IF
		END_IF

	(**** PUMP 2 ****)
	PUMP2_STATUS:	(* Status and Fault *)
		Modbus.MB_Lock := TRUE;
		Modbus.MB_Query.SlaveAddress := Address2;
		Modbus.MB_Query.FunctionCode := 3;
		ModBus.MB_Query.Read_StartAddress := 201;
		ModBus.MB_Query.Read_Quantity := 2;
		ModBus.MB_Start := TRUE;

		state := PUMP2_DATA;

	PUMP2_DATA:	(* Pump data *)
		IF NOT ModBus.MB_Start THEN
			IF ModBus.MB_MASTER.bInterfaceError<>0 THEN
				state := ERROR_STATE;
			ELSE
				DataPump2.PumpStatus := ModBus.MB_Resp.Data[0];
				DataPump2.PumpFault	:= WORD_TO_BOOL(ModBus.MB_Resp.Data[1]);

				ModBus.MB_Query.Read_StartAddress := 210;
				ModBus.MB_Query.Read_Quantity := 12;
				ModBus.MB_Start := TRUE;

				state := PUMP2_ALARMS;
			END_IF
		END_IF

	PUMP2_ALARMS:
		IF NOT ModBus.MB_Start THEN
			IF ModBus.MB_MASTER.bInterfaceError<>0 THEN
				state := ERROR_STATE;
			ELSE
				DataPump2.PumpBoardTemp := WORD_TO_INT(ModBus.MB_Resp.Data[0]);
				DataPump2.PumpVoltage	:= ModBus.MB_Resp.Data[2];
				DataPump2.PumpCurrent	:= ModBus.MB_Resp.Data[3];
				DataPump2.PumpRPM		:= ModBus.MB_Resp.Data[5];
				DataPump2.PumpPower		:= ModBus.MB_Resp.Data[6];
				DataPump2.PumpOpTime	:= BUILD_16TO32(ADR(ModBus.MB_Resp.Data[7]));
				DataPump2.PumpHead		:= ModBus.MB_Resp.Data[9];
				DataPump2.PumpFlow		:= ModBus.MB_Resp.Data[10];
				DataPump2.PumpLiqTemp	:= WORD_TO_INT(ModBus.MB_Resp.Data[11]);


				ModBus.MB_Query.Read_StartAddress := 230;
				ModBus.MB_Query.Read_Quantity := 15;
				ModBus.MB_Start := TRUE;

				state := PUMP2_END_READ;
			END_IF
		END_IF

	PUMP2_END_READ:
		IF NOT ModBus.MB_Start THEN
			IF ModBus.MB_MASTER.bInterfaceError<>0 THEN
				state := ERROR_STATE;
			ELSE
				DataPump2.PumpAlarm[0] := ModBus.MB_Resp.Data[0];
				DataPump2.PumpAlarm[1] := ModBus.MB_Resp.Data[1];
				DataPump2.PumpAlarm[2] := ModBus.MB_Resp.Data[2];
				DataPump2.PumpAlarm[3] := ModBus.MB_Resp.Data[3];
				DataPump2.PumpAlarm[4] := ModBus.MB_Resp.Data[4];
				DataPump2.PumpAlarm[5] := ModBus.MB_Resp.Data[5];
				DataPump2.PumpAlarm[6] := ModBus.MB_Resp.Data[6];
				DataPump2.PumpAlarm[7] := ModBus.MB_Resp.Data[7];
				DataPump2.PumpAlarm[8] := ModBus.MB_Resp.Data[8];
				DataPump2.PumpAlarm[9] := ModBus.MB_Resp.Data[9];
				DataPump2.PumpAlarm[10] := ModBus.MB_Resp.Data[10];
				DataPump2.PumpAlarm[11] := ModBus.MB_Resp.Data[11];
				DataPump2.PumpAlarm[12] := ModBus.MB_Resp.Data[12];
				DataPump2.PumpAlarm[13] := ModBus.MB_Resp.Data[13];
				DataPump2.PumpAlarm[14] := ModBus.MB_Resp.Data[14];

				retry := 0;
				state := WAIT_STATE;
			END_IF
		END_IF

	(**** WRITE ON/OFF REGISTER AND VERIFY RIGHT SETTING ****)
	CIR_ON_OFF:	(* Pump On/off *)
		Modbus.MB_Lock := TRUE;
		Modbus.MB_Query.SlaveAddress := Address1;
		Modbus.MB_Query.FunctionCode := 6;
		ModBus.MB_Query.Write_StartAddress := 110;
		ModBus.MB_Query.Write_Quantity := 1;
		ModBus.MB_Query.Write_Data[0] := BYTE_TO_WORD(CirStatus);
		ModBus.MB_Start := TRUE;

		state := CIR_ON_OFF_CHECK;

	CIR_ON_OFF_CHECK:	(* Check if write has been done correctly *)
		IF NOT ModBus.MB_Start THEN
			IF ModBus.MB_MASTER.bInterfaceError<>0 THEN
				state := ERROR_STATE;
			ELSE
				Modbus.MB_Query.SlaveAddress := Address1;
				Modbus.MB_Query.FunctionCode := 3;
				ModBus.MB_Query.Read_StartAddress := 110;
				ModBus.MB_Query.Read_Quantity := 1;
				ModBus.MB_Start := TRUE;

				state := CIR_END_WRITE;
			END_IF
		END_IF

	CIR_END_WRITE:
		IF NOT ModBus.MB_Start THEN
			IF ModBus.MB_MASTER.bInterfaceError<>0 THEN
				state := ERROR_STATE;
			ELSE
				IF ModBus.MB_Resp.Data[0] <> BYTE_TO_WORD(CirStatus) THEN
					state := CIR_ON_OFF;

					IF retry_write = 3 THEN
						LogEv(EL_Alarm,EO_CIRD,ID,28,'Modbus_write_error');
						Status_Log := 2;
						state := WAIT_STATE;
						retry_write := 0;
					ELSE
						retry_write := retry_write + 1;
					END_IF
				ELSE
					retry_write := 0;
					state := WAIT_STATE;
				END_IF
			END_IF
		END_IF


	(**** CHECK MODBUS ERROR ****)
	ERROR_STATE: 	(* Release MODBUS *)
			MODBUS.MB_Lock:=FALSE;

			(* Retries *)
			retry:=retry+1;
			IF retry>3 THEN
				retry:=0;
				(* Signal event *)
				IF Status_Log<>2 THEN
					LogEv(EL_Alarm,EO_CIRD,ID,27,'Modbus_communication_error');
				END_IF

				(* Update status *)
				Status_Log:=2;
				Status_Vis:=COLOR_RED;
			END_IF

			state:=WAIT_STATE;
END_CASE
END_ACTION

(* POU Plant_Objects/obj_MODBUS_CIR_DOPPIO_new, ST *)
FUNCTION_BLOCK obj_MODBUS_CIR_DOPPIO_new
VAR CONSTANT
	WAIT_STATE		:	BYTE := 0;
	PUMP1_STATUS	:	BYTE := 1;
	PUMP1_DATA		:	BYTE := 2;
	PUMP1_ALARMS	:	BYTE := 3;
	PUMP1_END_READ	:	BYTE := 4;
	PUMP2_STATUS	:	BYTE := 5;
	PUMP2_DATA		:	BYTE := 6;
	PUMP2_ALARMS	:	BYTE := 7;
	PUMP2_END_READ	:	BYTE := 8;
	CIR_ON_OFF1		:	BYTE := 90;
	CIR_ON_OFF2		:	BYTE := 91;
	CIR_ON_OFF_CHECK:	BYTE := 92;
	CIR_END_WRITE	:	BYTE := 93;
	ERROR_STATE		:	BYTE := 100;

END_VAR
VAR_INPUT
	ID		:	BYTE;
	Address1:	BYTE;		(* Pump 1 Modbus address *)
	Address2:	BYTE;		(* Pump 2 Modbus address *)

	(* Physical inputs (Force) *)
	CIR_RUN_REQ		: BOOL; (* External run request (no heat or cold requested) *)
	CIR_STOP_REQ	: BOOL; (* External stop request (has priority over RUN signals!) *)

	(* Physical inputs (Feedback) *)
	PumpA_AL		: BOOL; (* Alarm input signal *)
	PumpB_AL		: BOOL;
	PumpA_AUTO		: BOOL;	(* Automatic/Manual input *)
	PumpB_AUTO		: BOOL;

	(* Controls *)
	OnOff		: 	BOOL;	(* On/Off from chrono *)
	Mode		:	BYTE;	(* Working mode: 0-Both pumps works simultaneously, 1-Alternate every 24h, 2-Master/Backup *)
	InitOK		:	BOOL;

	(* Timings *)
	OnDelay		:	TIME;	(* Switch on delay *)
	OffDelay	:	TIME;	(* Switch off delay *)

	(* Modbus *)
	Refresh_Now	:	BOOL;	(* Start immediately modbus state machine *)
END_VAR
VAR_IN_OUT
	ModBus		:	obj_MODBUS;
END_VAR
VAR_OUTPUT
	Ctrl_Run	:	BOOL;		(* Logical status of the device: 0: Not running (switched off), 1: running *)
	Run			:	BOOL;		(* Real status *)

	Status_Log	:	WORD;
	Status_Vis	:	DWORD;
END_VAR
VAR
	Pump_En		:	ARRAY [1..2] OF BOOL;		(* Pumps enable *)

	ChangeTmr	: 	TON := (PT:=T#24h);			(* Timer that counts change time when in alternate mode *)
	ActivePump	: 	BYTE;						(* Actual active pump *)
	NewActivePump	: BYTE;

	(* Filters *)
	fPump_AL	: 	ARRAY [1..2] OF FLT_EVENT := (INITEV:=FALSE);
	fPump_ST	: 	ARRAY [1..2] OF FLT_EVENT := (INITEV:=FALSE);
	fPump_En	:	ARRAY [1..2] OF FLT_EVENT;
	fCIR_AUTO	:	ARRAY [1..2] OF FLT_EVENT;
	fStatusFault:	ARRAY [1..2] OF BOOL;

	(* Timer manage switch on/off delay *)
	Delay		: 	TONOF;

	(* CIR data structure *)
	DataPump1	:	typ_MODBUS_CIR;
	DataPump2	:	typ_MODBUS_CIR;

	(* Modbus variables *)
	state		:	BYTE;
	retry		:	BYTE;
	ReadTmr		:	TON := (PT:=T#5m);
	fModbusAlr	: 	BOOL;
	fWrite		:	ARRAY [1..2] OF BOOL;

	(* Alarm and Warning counters *)
	AlarmCtr	:	BYTE;
	WarningCtr	:	BYTE;

	(* Filers on alarms and faults *)
	AlarmHw		:	ARRAY [1..2] OF FLT_EVENT := (INITEV:=FALSE);
	Alarm		:	ARRAY [1..2] OF FLT_EVENT := (INITEV:=FALSE);
	Inverter	:	ARRAY [1..2] OF FLT_EVENT := (INITEV:=FALSE);
	ModbusAlr	:	FLT_EVENT := (INITEV:=FALSE);

	OldAlarmPump1	:	WORD;
	OldAlarmPump2	:	WORD;

END_VAR
Init();

PumpManager();

(* State machine to read pump parameters *)
Stm();

(* Check alarm and warning for both pumps *)
CheckFault();

(* Set output according to logical On/Off status *)
IF AlarmCtr>0 THEN Run := FALSE;
ELSE Run := Ctrl_Run;
END_IF

IF AlarmCtr>0 THEN
	Status_Log := 2;
	Status_Vis := COLOR_RED;
ELSIF WarningCtr>0 THEN
	Status_Log := 1;
	Status_Vis := COLOR_YELLOW;
ELSE
	Status_Log := 0;
	Status_Vis := COLOR_GREEN;
END_IF

(* Update error lamp status *)
Lamp.UpdateStatus(obj_Status := Status_Log);
END_FUNCTION_BLOCK
ACTION AddLogData:
Logger.s1:=INSERT('&CIR=',BYTE_TO_STRING(ID),4);
IF ID<10 THEN Logger.s1:=INSERT(Logger.s1,'0',4); END_IF

(* PUMP 1 *)
Logger.s1:=CONCAT(Logger.s1,WORD_TO_STRING(DataPump1.PumpStatus));		Logger.s1:=CONCAT(Logger.s1,';');
Logger.s1:=CONCAT(Logger.s1,INT_TO_STRING(DataPump1.PumpBoardTemp));	Logger.s1:=CONCAT(Logger.s1,';');
Logger.s1:=CONCAT(Logger.s1,WORD_TO_STRING(DataPump1.PumpVoltage));		Logger.s1:=CONCAT(Logger.s1,';');
Logger.s1:=CONCAT(Logger.s1,WORD_TO_STRING(DataPump1.PumpRPM));			Logger.s1:=CONCAT(Logger.s1,';');
Logger.s1:=CONCAT(Logger.s1,WORD_TO_STRING(DataPump1.PumpPower));		Logger.s1:=CONCAT(Logger.s1,';');
Logger.s1:=CONCAT(Logger.s1,DWORD_TO_STRING(DataPump1.PumpOpTime));		Logger.s1:=CONCAT(Logger.s1,';');
Logger.s1:=CONCAT(Logger.s1,WORD_TO_STRING(DataPump1.PumpHead));		Logger.s1:=CONCAT(Logger.s1,';');
Logger.s1:=CONCAT(Logger.s1,WORD_TO_STRING(DataPump1.PumpFlow));		Logger.s1:=CONCAT(Logger.s1,';');
Logger.s1:=CONCAT(Logger.s1,WORD_TO_STRING(DataPump1.PumpLiqTemp));		Logger.s1:=CONCAT(Logger.s1,';');

(* PUMP 2 *)
Logger.s1:=CONCAT(Logger.s1,WORD_TO_STRING(DataPump2.PumpStatus));		Logger.s1:=CONCAT(Logger.s1,';');
Logger.s1:=CONCAT(Logger.s1,INT_TO_STRING(DataPump2.PumpBoardTemp));	Logger.s1:=CONCAT(Logger.s1,';');
Logger.s1:=CONCAT(Logger.s1,WORD_TO_STRING(DataPump2.PumpVoltage));		Logger.s1:=CONCAT(Logger.s1,';');
Logger.s1:=CONCAT(Logger.s1,WORD_TO_STRING(DataPump2.PumpRPM));			Logger.s1:=CONCAT(Logger.s1,';');
Logger.s1:=CONCAT(Logger.s1,WORD_TO_STRING(DataPump2.PumpPower));		Logger.s1:=CONCAT(Logger.s1,';');
Logger.s1:=CONCAT(Logger.s1,DWORD_TO_STRING(DataPump2.PumpOpTime));		Logger.s1:=CONCAT(Logger.s1,';');
Logger.s1:=CONCAT(Logger.s1,WORD_TO_STRING(DataPump2.PumpHead));		Logger.s1:=CONCAT(Logger.s1,';');
Logger.s1:=CONCAT(Logger.s1,WORD_TO_STRING(DataPump2.PumpFlow));		Logger.s1:=CONCAT(Logger.s1,';');
Logger.s1:=CONCAT(Logger.s1,WORD_TO_STRING(DataPump2.PumpLiqTemp));		Logger.s1:=CONCAT(Logger.s1,';');

Logger.s1:=CONCAT(Logger.s1,WORD_TO_STRING(Status_Log));
ADDSTRING(ADR(Logger.TData), ADR(Logger.s1), Logger.TLen);
END_ACTION
ACTION CheckFault:
(*** WARNINGS ***)

(* Verify ModBus error	*)
ModbusAlr(IN:=fModbusAlr);

IF ModbusAlr.EVH THEN
	LogEv(EL_Wrn,EO_CIRD,ID,23,SEL(ModBus.MB_MASTER.MB_Error<>0,'0','1'));
	WarningCtr := WarningCtr + 1;
END_IF

IF ModbusAlr.EVL THEN WarningCtr := WarningCtr - 1; END_IF


(*** ALARMS ***)

(**** PUMP 1 ****)

(* Hardware alarm (physical input *)
AlarmHw[1](IN:=PumpA_AL);

IF AlarmHw[1].EVH THEN
	LogEv(EL_Alarm,EO_CIRD,ID,3,'CIR_Alarm_A');
	AlarmCtr := AlarmCtr + 1;
END_IF

IF AlarmHw[1].EVL THEN
	LogEv(EL_Log,EO_CIRD,ID,4,'CIR_Alarm_A_Recovered');
	AlarmCtr := AlarmCtr - 1;
END_IF

(* General alarm (read by Modbus) *)
Alarm[1](IN:=(DataPump1.PumpAlarm[0] <> OldAlarmPump1));

IF Alarm[1].EVH THEN
	IF DataPump1.PumpAlarm[1] = 0 THEN
		LogEv(EL_Alarm,EO_CIRD,ID,18,'Alarm_A_Recovered');
		AlarmCtr := AlarmCtr - 1;
	ELSE
		LogEv(EL_Alarm,EO_CIRD,ID,17,WORD_TO_STRING(DataPump1.PumpAlarm[1]));
		AlarmCtr := AlarmCtr + 1;
	END_IF

	OldAlarmPump1 := DataPump1.PumpAlarm[1];
END_IF

(* Inverter pump error *)
Inverter[1](IN:=DataPump1.PumpFault);

IF Inverter[1].EVH THEN
	LogEv(EL_Alarm,EO_CIRD,ID,15,'Inverter_Fault_A');
	AlarmCtr := AlarmCtr + 1;
END_IF

IF Inverter[1].EVL THEN
	LogEv(EL_Alarm,EO_CIRD,ID,16,'Inverter_Fault_A_Recovered');
	AlarmCtr := AlarmCtr - 1;
END_IF


(**** PUMP 2 ****)

(* Hardware alarm (physical input *)
AlarmHw[2](IN:=PumpB_AL);

IF AlarmHw[2].EVH THEN
	LogEv(EL_Alarm,EO_CIRD,ID,11,'CIR_Alarm_B');
	AlarmCtr := AlarmCtr + 1;
END_IF

IF AlarmHw[2].EVL THEN
	LogEv(EL_Log,EO_CIRD,ID,12,'CIR_Alarm_B_Recovered');
	AlarmCtr := AlarmCtr - 1;
END_IF

(* General alarm (read by Modbus) *)
Alarm[2](IN:=(DataPump2.PumpAlarm[0] <> OldAlarmPump2));

IF Alarm[2].EVH THEN
	IF DataPump2.PumpAlarm[0] = 0 THEN
		LogEv(EL_Log,EO_CIRD,ID,22,'Alarm_B_Recovered');
		AlarmCtr := AlarmCtr - 1;
	ELSE
		LogEv(EL_Alarm,EO_CIRD,ID,21,WORD_TO_STRING(DataPump2.PumpAlarm[0]));
		AlarmCtr := AlarmCtr + 1;
	END_IF

	OldAlarmPump2 := DataPump2.PumpAlarm[0];
END_IF

(* Inverter pump error *)
Inverter[2](IN:=DataPump2.PumpFault);

IF Inverter[2].EVH THEN
	LogEv(EL_Alarm,EO_CIRD,ID,19,'Inverter_Fault_B');
	AlarmCtr := AlarmCtr + 1;
END_IF

IF Inverter[2].EVL THEN
	LogEv(EL_Log,EO_CIRD,ID,20,'Inverter_Fault_B_Recovered');
	AlarmCtr := AlarmCtr - 1;
END_IF
END_ACTION
ACTION Init:
IF NOT InitOK THEN

	Delay.PT_OF := SEL(OffDelay=T#0s, OffDelay, Plant_CirOffDelay);
	Delay.PT_ON := SEL(OffDelay=T#0s, OnDelay, Plant_CirOnDelay) + WORD_TO_TIME(1000*ID);

	ReadTmr.PT := WORD_TO_TIME(1000*ID);	(* 1s delay between reads of 2 different double CIRs *)

	InitOK := TRUE;

END_IF
END_ACTION
ACTION PumpManager:
(*** Verify Status ***)
IF (Pump_En[1] AND DataPump1.PumpStatus=0) OR (NOT Pump_En[1] AND DataPump1.PumpStatus=2) THEN fStatusFault[1] := TRUE;
ELSE fStatusFault[1] := FALSE;
END_IF

IF (Pump_En[2] AND DataPump2.PumpStatus=0) OR (NOT Pump_En[2] AND DataPump2.PumpStatus=2) THEN fStatusFault[2] := TRUE;
ELSE fStatusFault[2] := FALSE;
END_IF

fPump_ST[1](IN:=fStatusFault[1]);
fPump_ST[2](IN:=fStatusFault[2]);

IF fPump_ST[1].EVH THEN
	LogEv(SEL(Pump_En[1],EL_Alarm,EL_Wrn),EO_CIRD,ID,SEL(Pump_En[1],5,6),'');
	WarningCtr := WarningCtr + 1;
END_IF

IF fPump_ST[1].EVL THEN WarningCtr := WarningCtr - 1; END_IF

IF fPump_ST[2].EVH THEN
	LogEv(SEL(Pump_En[2],EL_Alarm,EL_Wrn),EO_CIRD,ID,SEL(Pump_En[2],13,14),'');
	WarningCtr := WarningCtr + 1;
END_IF

IF fPump_ST[2].EVL THEN WarningCtr := WarningCtr - 1; END_IF


(* Verify if in Auto or Manual mode *)
fCIR_AUTO[1](IN:=PumpA_AUTO);
fCIR_AUTO[2](IN:=PumpB_AUTO);

(*** Pump A ***)
IF fCIR_AUTO[1].EVH THEN
	LogEv(EL_Log,EO_CIRD,ID,8,'CIR_Auto');
	WarningCtr := WarningCtr - 1;
END_IF

(* Manual -> Keep switched on *)
IF fCIR_AUTO[1].EVL THEN
	LogEv(EL_Wrn,EO_CIRD,ID,7,'CIR_Manual');
	WarningCtr := WarningCtr + 1;

	(* Switch on pump A *)
	Pump_En[1] := 0;
END_IF

(*** Pump B ***)
IF fCIR_AUTO[2].EVH THEN
	LogEv(EL_Log,EO_CIRD,ID,8,'CIR_Auto');
	WarningCtr := WarningCtr - 1;
END_IF

(* Manual -> Keep switched on *)
IF fCIR_AUTO[2].EVL THEN
	LogEv(EL_Wrn,EO_CIRD,ID,7,'CIR_Manual');
	WarningCtr := WarningCtr + 1;

	(* Switch on pump B *)
	Pump_En[2] := 0;
END_IF

(* If working mode is Alternate, count change time *)
ChangeTmr(IN:=(Mode=1));

IF ChangeTmr.Q THEN

	NewActivePump := SEL(ActivePump=1,1,2);

	(* If no alarm on other pump, keep going with the switch *)
	IF NOT fPump_AL[NewActivePump].IN THEN	ActivePump := NewActivePump;
	ELSE LogEv(EL_Wrn,EO_CIRD,ID,29,'');		(* Pump not switched because of other pump's failure *)
	END_IF

	(* Switch off "old" working pump and on "new" working one *)
	Pump_En[1] := SEL(ActivePump=1,TRUE,FALSE);
	Pump_En[2] := SEL(ActivePump=1,FALSE,TRUE);

	fWrite[1] := TRUE;
	fWrite[2] := TRUE;

	ChangeTmr.PT:=T#24h;
END_IF

(* Verify if OnOff is changed *)
Ctrl_Run := OnOff;

(* Check switch on or switch off delay *)
Delay(IN:=Ctrl_Run);

(* Set output according to actual function mode *)
CASE Mode OF

	0:	(*** Simultaneous pumps working ***)
		IF CIR_STOP_REQ THEN
			Pump_En[1] := SEL(PumpA_AUTO,FALSE,TRUE);
			Pump_En[2] := SEL(PumpB_AUTO,FALSE,TRUE);
		ELSIF CIR_RUN_REQ THEN
			Pump_En[1] := 0;
			Pump_En[2] := 0;
		ELSE
			Pump_En[1] := SEL(PumpA_AUTO,FALSE,NOT Delay.OUT);
			Pump_En[2] := SEL(PumpB_AUTO,FALSE,NOT Delay.OUT);
		END_IF

		(* Set RUN signal (for external objects) *)
		IF fPump_AL[1].IN OR fPump_AL[2].IN OR fPump_ST[1].IN OR fPump_ST[2].IN THEN
			Ctrl_Run:=FALSE;
		ELSE
			Run:=Delay.OUT;
		END_IF

	1,2:  (*** Alternate working and Master/backup mode ***)
		IF fPump_AL[ActivePump].IN THEN
			ActivePump := SEL(ActivePump=1,1,2);
			LogEv(EL_Wrn,EO_CIRD,ID,30,'');	(* Pump switched because of current pump failure *)

			(* Switch off alarm pump and on "new" working one *)
			Pump_En[1] := SEL(ActivePump=1,TRUE,FALSE);
			Pump_En[2] := SEL(ActivePump=1,FALSE,TRUE);
		
			fWrite[1] := TRUE;
			fWrite[2] := TRUE;
		END_IF

		IF fCIR_AUTO[ActivePump].IN THEN
			(* If priority request *)
			IF CIR_STOP_REQ THEN
				Pump_En[ActivePump] := 1;
			ELSIF CIR_RUN_REQ THEN
				Pump_En[ActivePump] := 0;
			ELSE
				Pump_En[ActivePump] := NOT Delay.OUT;
			END_IF
	
			(* Set RUN signal (for external objects) *)
			IF fPump_AL[ActivePump].IN OR fPump_ST[ActivePump].IN THEN
				Ctrl_Run:=FALSE;
			ELSE
				Run:=Delay.OUT;
			END_IF
		END_IF

END_CASE

(* Check if a pump enable update (modbus write) is requested *)
fPump_En[1](IN:=Pump_En[1]);
fPump_En[2](IN:=Pump_En[2]);

IF fPump_En[1].EVH OR fPump_En[1].EVL THEN
	fWrite[1] := TRUE;
	Refresh_Now := TRUE;
END_IF
IF fPump_En[2].EVH OR fPump_En[2].EVL THEN
	fWrite[2] := TRUE;
	Refresh_Now := TRUE;
END_IF
END_ACTION
ACTION Stm:
CASE state OF
	WAIT_STATE:	(* Refresh time manager *)
		ReadTmr(IN:=NOT ReadTmr.Q);
		IF ReadTmr.Q OR Refresh_Now THEN
			state := PUMP1_STATUS;
			ReadTmr.PT := T#1m;
			Refresh_Now := FALSE;
		END_IF

	(**** READ CIR PARAMETERS ****)

	(**** PUMP 1 ****)
	PUMP1_STATUS:	(* Status and Fault *)
		Modbus.MB_Lock := TRUE;

		Modbus.MB_Query.SlaveAddress := Address1;
		Modbus.MB_Query.FunctionCode := 3;
		ModBus.MB_Query.Read_StartAddress := 201;
		ModBus.MB_Query.Read_Quantity := 2;
		ModBus.MB_Start := TRUE;

		state := PUMP1_DATA;

	PUMP1_DATA:	(* Pump data *)
		IF NOT ModBus.MB_Start THEN
			IF ModBus.MB_MASTER.bInterfaceError<>0 OR ModBus.MB_MASTER.MB_Error<>0 THEN
				state := ERROR_STATE;
			ELSE
				DataPump1.PumpStatus := ModBus.MB_Resp.Data[0];
				DataPump1.PumpFault	:= WORD_TO_BOOL(ModBus.MB_Resp.Data[1]);

				ModBus.MB_Query.Read_StartAddress := 210;
				ModBus.MB_Query.Read_Quantity := 12;
				ModBus.MB_Start := TRUE;

				state := PUMP1_ALARMS;
			END_IF
		END_IF

	PUMP1_ALARMS: (* Historical alarms *)
		IF NOT ModBus.MB_Start THEN
			IF ModBus.MB_MASTER.bInterfaceError<>0 OR ModBus.MB_MASTER.MB_Error<>0  THEN
				state := ERROR_STATE;
			ELSE
				DataPump1.PumpBoardTemp := WORD_TO_INT(ModBus.MB_Resp.Data[0]);
				DataPump1.PumpVoltage	:= ModBus.MB_Resp.Data[2];
				DataPump1.PumpCurrent	:= ModBus.MB_Resp.Data[3];
				DataPump1.PumpRPM		:= ModBus.MB_Resp.Data[5];
				DataPump1.PumpPower		:= ModBus.MB_Resp.Data[6];
				DataPump1.PumpOpTime	:= BUILD_16TO32(ADR(ModBus.MB_Resp.Data[7]));
				DataPump1.PumpHead		:= ModBus.MB_Resp.Data[9];
				DataPump1.PumpFlow		:= ModBus.MB_Resp.Data[10];
				DataPump1.PumpLiqTemp	:= WORD_TO_INT(ModBus.MB_Resp.Data[11]);


				ModBus.MB_Query.Read_StartAddress := 230;
				ModBus.MB_Query.Read_Quantity := 15;
				ModBus.MB_Start := TRUE;

				state := PUMP1_END_READ;
			END_IF
		END_IF

	PUMP1_END_READ:	(* Read alarms *)
		IF NOT ModBus.MB_Start THEN
			IF ModBus.MB_MASTER.bInterfaceError<>0 OR ModBus.MB_MASTER.MB_Error<>0  THEN
				state := ERROR_STATE;
			ELSE
				DataPump1.PumpAlarm[0] := ModBus.MB_Resp.Data[0];
				DataPump1.PumpAlarm[1] := ModBus.MB_Resp.Data[1];
				DataPump1.PumpAlarm[2] := ModBus.MB_Resp.Data[2];
				DataPump1.PumpAlarm[3] := ModBus.MB_Resp.Data[3];
				DataPump1.PumpAlarm[4] := ModBus.MB_Resp.Data[4];
				DataPump1.PumpAlarm[5] := ModBus.MB_Resp.Data[5];
				DataPump1.PumpAlarm[6] := ModBus.MB_Resp.Data[6];
				DataPump1.PumpAlarm[7] := ModBus.MB_Resp.Data[7];
				DataPump1.PumpAlarm[8] := ModBus.MB_Resp.Data[8];
				DataPump1.PumpAlarm[9] := ModBus.MB_Resp.Data[9];
				DataPump1.PumpAlarm[10] := ModBus.MB_Resp.Data[10];
				DataPump1.PumpAlarm[11] := ModBus.MB_Resp.Data[11];
				DataPump1.PumpAlarm[12] := ModBus.MB_Resp.Data[12];
				DataPump1.PumpAlarm[13] := ModBus.MB_Resp.Data[13];
				DataPump1.PumpAlarm[14] := ModBus.MB_Resp.Data[14];

				state := PUMP2_STATUS;
			END_IF
		END_IF

	(**** PUMP 2 ****)
	PUMP2_STATUS:	(* Status and Fault *)
		Modbus.MB_Lock := TRUE;
		Modbus.MB_Query.SlaveAddress := Address2;
		Modbus.MB_Query.FunctionCode := 3;
		ModBus.MB_Query.Read_StartAddress := 201;
		ModBus.MB_Query.Read_Quantity := 2;
		ModBus.MB_Start := TRUE;

		state := PUMP2_DATA;

	PUMP2_DATA:	(* Pump data *)
		IF NOT ModBus.MB_Start THEN
			IF ModBus.MB_MASTER.bInterfaceError<>0 OR ModBus.MB_MASTER.MB_Error<>0  THEN
				state := ERROR_STATE;
			ELSE
				DataPump2.PumpStatus := ModBus.MB_Resp.Data[0];
				DataPump2.PumpFault	:= WORD_TO_BOOL(ModBus.MB_Resp.Data[1]);

				ModBus.MB_Query.Read_StartAddress := 210;
				ModBus.MB_Query.Read_Quantity := 12;
				ModBus.MB_Start := TRUE;

				state := PUMP2_ALARMS;
			END_IF
		END_IF

	PUMP2_ALARMS:
		IF NOT ModBus.MB_Start THEN
			IF ModBus.MB_MASTER.bInterfaceError<>0 OR ModBus.MB_MASTER.MB_Error<>0  THEN
				state := ERROR_STATE;
			ELSE
				DataPump2.PumpBoardTemp := WORD_TO_INT(ModBus.MB_Resp.Data[0]);
				DataPump2.PumpVoltage	:= ModBus.MB_Resp.Data[2];
				DataPump2.PumpCurrent	:= ModBus.MB_Resp.Data[3];
				DataPump2.PumpRPM		:= ModBus.MB_Resp.Data[5];
				DataPump2.PumpPower		:= ModBus.MB_Resp.Data[6];
				DataPump2.PumpOpTime	:= BUILD_16TO32(ADR(ModBus.MB_Resp.Data[7]));
				DataPump2.PumpHead		:= ModBus.MB_Resp.Data[9];
				DataPump2.PumpFlow		:= ModBus.MB_Resp.Data[10];
				DataPump2.PumpLiqTemp	:= WORD_TO_INT(ModBus.MB_Resp.Data[11]);


				ModBus.MB_Query.Read_StartAddress := 230;
				ModBus.MB_Query.Read_Quantity := 15;
				ModBus.MB_Start := TRUE;

				state := PUMP2_END_READ;
			END_IF
		END_IF

	PUMP2_END_READ:
		IF NOT ModBus.MB_Start THEN
			IF ModBus.MB_MASTER.bInterfaceError<>0 OR ModBus.MB_MASTER.MB_Error<>0  THEN
				state := ERROR_STATE;
			ELSE
				DataPump2.PumpAlarm[0] := ModBus.MB_Resp.Data[0];
				DataPump2.PumpAlarm[1] := ModBus.MB_Resp.Data[1];
				DataPump2.PumpAlarm[2] := ModBus.MB_Resp.Data[2];
				DataPump2.PumpAlarm[3] := ModBus.MB_Resp.Data[3];
				DataPump2.PumpAlarm[4] := ModBus.MB_Resp.Data[4];
				DataPump2.PumpAlarm[5] := ModBus.MB_Resp.Data[5];
				DataPump2.PumpAlarm[6] := ModBus.MB_Resp.Data[6];
				DataPump2.PumpAlarm[7] := ModBus.MB_Resp.Data[7];
				DataPump2.PumpAlarm[8] := ModBus.MB_Resp.Data[8];
				DataPump2.PumpAlarm[9] := ModBus.MB_Resp.Data[9];
				DataPump2.PumpAlarm[10] := ModBus.MB_Resp.Data[10];
				DataPump2.PumpAlarm[11] := ModBus.MB_Resp.Data[11];
				DataPump2.PumpAlarm[12] := ModBus.MB_Resp.Data[12];
				DataPump2.PumpAlarm[13] := ModBus.MB_Resp.Data[13];
				DataPump2.PumpAlarm[14] := ModBus.MB_Resp.Data[14];

				IF fModbusAlr THEN fModbusAlr := FALSE; END_IF

				IF fWrite[1] THEN state := CIR_ON_OFF1;
				ELSIF fWrite[2] THEN state := CIR_ON_OFF2;
				ELSE
					ModBus.MB_Lock := FALSE;
					retry := 0;
					state := WAIT_STATE;
				END_IF
			END_IF
		END_IF

	(**** WRITE ON/OFF REGISTER AND VERIFY RIGHT SETTING ****)

	CIR_ON_OFF1:	(* Pump A On/off *)

		Modbus.MB_Query.SlaveAddress := Address1;
		Modbus.MB_Query.FunctionCode := 6;
		ModBus.MB_Query.Write_StartAddress := 110;
		ModBus.MB_Query.Write_Quantity := 1;
		ModBus.MB_Query.Write_Data[0] := BOOL_TO_WORD(Pump_En[1]);
		ModBus.MB_Start := TRUE;

		IF fWrite[2] THEN state := CIR_ON_OFF2;
		ELSE state := CIR_END_WRITE;
		END_IF

	CIR_ON_OFF2:

	IF NOT ModBus.MB_Start THEN
		IF ModBus.MB_MASTER.bInterfaceError<>0 OR ModBus.MB_MASTER.MB_Error<>0  THEN
			state := ERROR_STATE;
		ELSE
			fWrite[1] := FALSE;

			Modbus.MB_Query.SlaveAddress := Address2;
			Modbus.MB_Query.FunctionCode := 6;
			ModBus.MB_Query.Write_StartAddress := 110;
			ModBus.MB_Query.Write_Quantity := 1;
			ModBus.MB_Query.Write_Data[0] := BOOL_TO_WORD(Pump_En[2]);
			ModBus.MB_Start := TRUE;

			state := CIR_END_WRITE;
		END_IF
	END_IF

	CIR_END_WRITE:
		IF NOT ModBus.MB_Start THEN
			IF ModBus.MB_MASTER.bInterfaceError<>0 OR ModBus.MB_MASTER.MB_Error<>0 THEN
				state := ERROR_STATE;
			ELSE
				fWrite[2] := FALSE;

				ModBus.MB_Lock := FALSE;
				retry := 0;
				state := WAIT_STATE;
			END_IF
		END_IF

	(**** CHECK MODBUS ERROR ****)
	ERROR_STATE: 	(* Release MODBUS *)
			MODBUS.MB_Lock:=FALSE;

			(* Retries *)
			retry:=retry+1;
			IF retry>3 THEN
				retry:=0;
				(* Signal event *)
				fModbusAlr := TRUE;
			END_IF

			state:=WAIT_STATE;
END_CASE
END_ACTION

(* POU Plant_Objects/obj_MODBUS_TCP, ST *)
FUNCTION_BLOCK obj_MODBUS_TCP
(* === MODBUS-TCP PROTOCOL INTERFACE ===
   v1.0[10/06/15] - Create
*)
VAR CONSTANT
	VARS_Max	: BYTE := 32;
END_VAR
VAR_INPUT
	(* Settings *)
	ID			: BYTE;
	IP			: STRING;
	PORT		: WORD:=502;
	(* Interface *)
	MB_MASTER	: ETHERNET_MODBUSMASTER_TCP;
	MB_READBUF	: ARRAY [0..128] OF WORD;
	MB_WRITEBUF : ARRAY [0..128] OF WORD;
	MB_Start	: BOOL;
	MB_Lock		: BOOL;
	(* Variables management *)
	VARS_En		: BOOL;
	VARS		: ARRAY [0..VARS_Max] OF typ_MODBUS_VAR;
	VARS_Check	: BOOL;
	VARS_Alarm	: BOOL;
	(* Variables allocation *)
	VAR_Pointer : POINTER TO ARRAY[0..99] OF WORD;
	VAR_Cfg		: POINTER TO typ_MODBUS_VAR;
END_VAR
VAR_OUTPUT
	(* Status *)
	Status_Log	: BYTE;
	Status_Vis	: DWORD;
END_VAR
VAR
	sta         : BYTE :=0;
	i			: BYTE;
	j			: BYTE;
	Alarm		: FLT_EVENT;

	VarTmr		: TON := (PT:=T#1s);
	VarSta		: BYTE; (* Status *)
	VarCnt		: BYTE; (* Scan counter *)
	VarRetry	: BYTE;
	VarAlarm	: BYTE; (* Last variable with errors *)
END_VAR
MB_MASTER( strIP_ADDRESS:=IP, wPORT:=PORT, tTIME_OUT:=T#750MS, (*xCONNECT:=TRUE,*)
		   ptREAD_DATA:=ADR(MB_READBUF), ptSEND_DATA:=ADR(MB_WRITEBUF), xSEND:=MB_Start );

IF sta=0 THEN
	MB_MASTER.xCONNECT:=TRUE;
	sta:=1;
END_IF

(* Process variable management *)
IF VARS_En THEN VARS_Process(); END_IF

(* Check status *)
Alarm(IN:=(MB_MASTER.wERROR<>0));
IF Alarm.EVH THEN
	LogEv(SEL(MB_MASTER.wERROR>0,EL_Wrn,EL_Alarm),EO_MODBUS_TCP,ID,1,WORD_TO_STRING(MB_MASTER.wERROR));
END_IF
IF Alarm.EVL THEN
	LogEv(EL_Log,EO_MODBUS_TCP,ID,2,'');
END_IF

(* Log/visu status *)
   IF Alarm.IN   THEN Status_Log:=2; Status_Vis:=COLOR_RED;
ELSIF Vars_Alarm THEN Status_Log:=1; Status_Vis:=COLOR_YELLOW;
  				 ELSE Status_Log:=0; Status_Vis:=COLOR_GREEN;
END_IF
END_FUNCTION_BLOCK
ACTION VAR_Search:
(* Search VAR with specific pointer if not found return first free VAR
	[Last VAR is not active... used as safe area...] 
*)
j:=VARS_Max;
FOR i := 0 TO VARS_Max-1 DO
	IF VARS[i].Variable=0 AND j>i THEN j:=i; END_IF
	IF VARS[i].Variable=VAR_Pointer THEN
		VAR_Cfg:=ADR(VARS[i]);
		RETURN;
	END_IF
END_FOR
VAR_Cfg:=ADR(VARS[j]);
END_ACTION
ACTION VARS_Process:
(* Update var timers *)
VarTmr(IN:=(NOT VarTmr.Q));
IF VarTmr.Q THEN
	FOR i := 0 TO VARS_Max DO
		IF VARS[i].Refresh_Cnt>0 THEN VARS[i].Refresh_Cnt:=VARS[i].Refresh_Cnt-1; END_IF
	END_FOR
	VARS_Check:=TRUE;
END_IF


(* Process status *)
CASE VarSta OF
	0: (* === Init *)
		VarCnt:=0;
		VarSta:=1;

	1: (* === Wait check signal *)
		IF VARS_Check THEN
			VARS_Check:=FALSE;
			VarCnt:=0;
			VarSta:=2;
		END_IF

	2: (* === Check loop *)
		IF NOT (MB_Lock OR MB_Start) THEN
			WHILE VarCnt<=(VARS_Max-1) AND VarSta=2 DO
				(* Check only active vars *)
				IF VARS[VarCnt].Variable<>0 THEN
					(* Check var auto-refresh on timer checks *)
					IF VARS[VarCnt].Refresh_Time>0 AND VARS[VarCnt].Refresh_Cnt=0 THEN
						VARS[VarCnt].Refresh_Cnt:=VARS[VarCnt].Refresh_Time;
						VarSta:=3;
					END_IF
					(* Check refresh for change or request *)
					CASE VARS[VarCnt].FunCode OF
						5,6,15,16: (* Write functions *)
							IF VARS[VarCnt].Variable_Size=1 THEN
								IF VARS[VarCnt].Variable^<>VARS[VarCnt].Variable_Mirror THEN
									VARS[VarCnt].Variable_Mirror:=VARS[VarCnt].Variable^;
									VarSta:=3;
								END_IF
							ELSE
								IF VARS[VarCnt].Variable_Mirror<>0 THEN
									VARS[VarCnt].Variable_Mirror:=0;
									VarSta:=3;
								END_IF
							END_IF
						1,2,3,4: (* Write functions *)
							IF VARS[VarCnt].Variable_Mirror<>0 THEN
								VARS[VarCnt].Variable_Mirror:=0;
								VarSta:=3;
							END_IF
					END_CASE
				END_IF
				(* Process query *)
				IF VarSta=3 THEN
					MB_Lock:=TRUE;
					MB_MASTER.bUNIT_ID:=VARS[VarCnt].SlaveAddress;
					MB_MASTER.bFUNCTION_CODE:=VARS[VarCnt].FunCode;
					CASE VARS[VarCnt].FunCode OF
						16#5,16#6,16#F,16#10:
							MB_MASTER.wREAD_ADDRESS:=0;
							MB_MASTER.wREAD_QUANTITY:=0;
							MB_MASTER.wWRITE_ADDRESS:=VARS[VarCnt].FunAddress;
							MB_MASTER.wWRITE_QUANTITY:=VARS[VarCnt].Variable_Size;
							IF VARS[VarCnt].Variable_Size=200 THEN
								COPY_32SWAP16(VARS[VarCnt].Variable, ADR(MB_WRITEBUF));
							ELSIF VARS[VarCnt].Variable_Size>1 THEN
								MEMCPY(VARS[VarCnt].Variable, ADR(MB_WRITEBUF), 2*VARS[VarCnt].Variable_Size);
							ELSE
								MB_WRITEBUF[0]:=VARS[VarCnt].Variable^;
							END_IF
						16#1,16#2,16#3,16#4:
							MB_MASTER.wREAD_ADDRESS:=VARS[VarCnt].FunAddress;
							IF VARS[VarCnt].Variable_Size=200 THEN MB_MASTER.wREAD_QUANTITY:=2; ELSE
							  MB_MASTER.wREAD_QUANTITY:=VARS[VarCnt].Variable_Size;
							END_IF
							MB_MASTER.wWRITE_ADDRESS:=0;
							MB_MASTER.wWRITE_QUANTITY:=0;
					END_CASE
					VarRetry:=0;
					MB_Start:=TRUE;
				ELSE
					VarCnt:=VarCnt+1;
				END_IF
			END_WHILE
			(* Check loop completed -> no actions *)
			IF VarSta=2 THEN VarSta:=1; END_IF
		END_IF

	3: (* === Wait & process MB response *)
		IF NOT MB_Start THEN
			IF MB_MASTER.wERROR=0 THEN
				CASE VARS[VarCnt].FunCode OF
					1,2,3,4:
						IF VARS[VarCnt].Variable_Size=200 THEN
							COPY_32SWAP16(ADR(MB_READBUF), VARS[VarCnt].Variable);
						ELSIF VARS[VarCnt].Variable_Size>1 THEN
							MEMCPY(ADR(MB_READBUF), VARS[VarCnt].Variable, 2*VARS[VarCnt].Variable_Size);
						ELSE
							VARS[VarCnt].Variable^:=MB_READBUF[0];
						END_IF
				END_CASE
				MB_Lock:=FALSE;
				(* Signal error recovery *)
				IF VARS_Alarm=TRUE AND VarCnt=VarAlarm THEN
					LogEv(EL_Wrn,EO_MODBUS_TCP,ID,5,'');
					VARS_Alarm:=FALSE;
				END_IF
				(* Next var *)
				VarCnt:=VarCnt+1;
				VarSta:=2;
			ELSE
				IF VarRetry<10 THEN
					VarRetry:=VarRetry+1;
					MB_Start:=TRUE;
				ELSE
					MB_Lock:=FALSE;
					(* Signal error *)
					IF VARS_Alarm=FALSE THEN
						LogEv(EL_Wrn,EO_MODBUS_TCP,ID,3,WORD_TO_STRING(MB_MASTER.wERROR));
						VARS_Alarm:=TRUE;
						VarAlarm:=VarCnt-1;
					END_IF
					(* Next var *)
					VarCnt:=VarCnt+1;
					VarSta:=2;
				END_IF
			END_IF
		END_IF

ELSE
	VarSta:=0;
END_CASE
END_ACTION

(* POU Plant_Objects/obj_TPV, ST *)
FUNCTION_BLOCK obj_TPV
(* === TEMPERATURE PROBE  ===
   v1.0[16/04/15] - Versioning
*)
VAR CONSTANT
	NormalEv		: BYTE := 0;
	ErrorEv			: BYTE := 1;
	WarningEv		: BYTE := 2;
END_VAR
VAR_INPUT
	(* Settings *)
	ID				: BYTE;
	TAP				: BYTE:=4;	   (* Consecutive checks filter *)
	INITEV			: BOOL:= TRUE; (* Generate init OK event *)
	IN_EMIN			: INT :=-2000; (* Low error limit *)
	IN_WMIN			: INT := -550; (* Low warning value *)
	IN_WMAX			: INT :=  900; (* High warning value *)
	IN_EMAX			: INT := 8500; (* High error limit *)
	ERR_MIN_SHORT	: BOOL:= TRUE; (* TRUE  ==> EMIN=Short        , EMAX=Disconnected
									  FALSE ==> EMIN=Disconnected , EMAX=Short 		 *)
	(* Physical input *)
	IN			: INT;
END_VAR
VAR_OUTPUT
	WRN			: BOOL;	(* Value in warning range *)
	ERR			: BOOL;	(* Value error *)
	HI			: INT;	(* Highest value - cleared by Stat_Reset() action *)
	AVG			: INT; 	(* Average value - updated by Mean() action, cleared by Mean_Reset() action *)
	LOW			: INT;	(* Lowest value  - cleared by Stat_Reset() action *)

	Status_Log	: WORD;
	Status_Vis	: DWORD;
END_VAR
VAR
	cnt			: BYTE;
	event		: BYTE := 0;	(* 0: monitoring a generic, 1: monitoring an error, 2: monitoring a warning *)
	asum		: DINT;
	acnt		: WORD;
END_VAR
(* Check probe value limits *)
IF IN<=IN_EMIN OR IN>=IN_EMAX THEN
	IF NOT ERR THEN
		IF event <> ErrorEv THEN
			cnt := 1;
			event := ErrorEv;
		ELSE
			cnt:=cnt+1;
		END_IF

		IF cnt>TAP THEN
			cnt:=0;
			ERR:=TRUE; WRN:=FALSE;
			IF ( ERR_MIN_SHORT=TRUE  AND IN<=IN_EMIN ) OR ( ERR_MIN_SHORT=FALSE AND IN>=IN_EMAX ) THEN
				LogEv(EL_Alarm,EO_TPV,ID,5,INT_TO_STRING(IN));
			ELSE
				LogEv(EL_Alarm,EO_TPV,ID,4,INT_TO_STRING(IN));
			END_IF
		END_IF
	END_IF
ELSIF IN<=IN_WMIN OR IN>=IN_WMAX THEN
	IF NOT WRN THEN
		IF event <> WarningEv THEN
			cnt := 1;
			event := WarningEv;
		ELSE
			cnt:=cnt+1;
		END_IF

		IF cnt>TAP THEN
			cnt:=0;
			ERR:=FALSE; WRN:=TRUE;
			LogEv(EL_Wrn,EO_TPV,ID,SEL(IN<=IN_WMIN,3,2),INT_TO_STRING(IN));
		END_IF
	END_IF
ELSE
	IF INITEV OR WRN OR ERR THEN
		IF event <> NormalEv THEN
			cnt := 1;
			event := NormalEv;
		ELSE
			cnt:=cnt+1;
		END_IF

		IF cnt>TAP THEN
			cnt:=0;
			INITEV:=FALSE; ERR:=FALSE; WRN:=FALSE;
			LogEv(EL_Log,EO_TPV,ID,1,'Probe_OK');
		END_IF
	END_IF
END_IF

(* Average value *)
IF acnt>=60000 THEN
	Mean();
	asum := asum - AVG;
	acnt := acnt - 1;
END_IF

asum := asum + IN;
acnt := acnt + 1;

(* Statistics values *)
IF IN<LOW THEN LOW:=IN; END_IF
IF IN>HI  THEN HI :=IN; END_IF

Lamp.obj_Status := Status_Log;
Lamp.UpdateStatus();

(* Status Log *)
IF ERR THEN	Status_Log := 2; Status_Vis := COLOR_RED;
ELSIF WRN THEN Status_Log := 1;	Status_Vis := COLOR_YELLOW;
ELSE Status_Log := 0; Status_Vis := COLOR_GREEN;
END_IF
END_FUNCTION_BLOCK
ACTION AddLogData:
Logger.s1:=INSERT('&TPV=',BYTE_TO_STRING(ID),4);
IF ID<10 THEN Logger.s1:=INSERT(Logger.s1,'0',4); END_IF

Mean();

Logger.s1:=CONCAT(Logger.s1,INT_TO_STRING(AVG));		Logger.s1:=CONCAT(Logger.s1,';');

Logger.s1:=CONCAT(Logger.s1,WORD_TO_STRING(Status_Log));
ADDSTRING(ADR(Logger.TData), ADR(Logger.s1), Logger.TLen);
END_ACTION
ACTION Mean:
AVG := DINT_TO_INT(asum/acnt);
END_ACTION
ACTION Mean_Reset:
AVG:=IN;
asum:=IN;
acnt:=1;
END_ACTION
ACTION Stat_Reset:
HI:=IN;
LOW:=IN;
END_ACTION

(* POU Plant_Objects/obj_VRD, ST *)
FUNCTION_BLOCK obj_VRD
(* === VALVOLA RIPARTITORE ===
   v1.0[16/04/15] - Versioning
*)
VAR_INPUT
	(* Settings *)
	ID				: BYTE;
	(* Controls *)
	RUN  			: BOOL;		(* Control input *)
	ReducedRange	: BOOL;		(* If true output value is among 2 and 10V, otherwise 0-10V *)

	(* Physical inputs *)
	TEMP 			: INT;		(* Input temperature from sensor *)
	STATUS 			: WORD;		(* Input position from valve *)

	InitOK			: BOOL;
	Alarm1			: BOOL;
	Alarm2			: BOOL;
	Warning			: BOOL;

	Ctrl_Init		: BOOL;
	Ctrl_SetPoint	: INT;
	Ctrl_Err		: INT;			(* Current error *)
	Ctrl_Err0		: INT; 			(* Previous error *)
	Ctrl_Accel		: REAL;			(* Derivate of error *)
	Ctrl_AccelGate  : INT:=1;		(* Derivate gate *)
	Ctrl_AccelTmr	: WORD;
	Ctrl_ErrGate	: INT:=1;		(* Error gate *)
	Ctrl_Kp			: REAL:=1;		(* Proportional factor *)
	Ctrl_Kd			: REAL:=100;  	(* Derivative factor *)
	Ctrl_Out		: REAL;

	Chk_Err			: INT;
	Chk_ErrGate		: INT:=20; 		(* Check error gate *)
	Chk_Cnt			: INT;
	Chk_CntAlarm	: INT:=60; 		(* Check error trigger 60s *)

	(* Status *)
	Log_AvgTemp		: AVERAGE_T;
	Status_Log		: BYTE;
	Status_Vis 		: DWORD;

END_VAR
VAR_IN_OUT
	CLIM		: typ_Clima;
END_VAR
VAR_OUTPUT
	(* Physical outputs *)
	OUT			: WORD;
END_VAR
VAR
	Curve		: CHARCURVE;
	Curve_Err	: BYTE;
END_VAR
(* Check initialization *)
(*IF NOT InitOK THEN Init(); END_IF*)

(* Check max temperature *)
IF TEMP>Plant_VRD_TAlarm THEN
	IF NOT Alarm1 THEN
		Alarm1:=TRUE;
		LogEv(EL_AlarmStop,EO_VRD,ID,3,'VRD_Overtemperature');
	END_IF
END_IF

(* Check climatic setup *)
IF NOT CLIM.InitOK THEN	DefaultClim(); END_IF;
(* Calculate Setpoint *)
Curve(	IN:= T_AMB,	N:= 5, P:= CLIM.Points,			(* Given the x value as input, the corresponding y value as output is returned, if it matches the crve designed by array of points *)
		OUT=> Ctrl_SetPoint, ERR=> Curve_Err );
IF Curve_Err>0 OR Ctrl_SetPoint>Plant_VRD_TMax THEN
	Ctrl_SetPoint:=Plant_VRD_TDefault;
	IF NOT Warning THEN
		Warning:=TRUE;
		LogEv(EL_Wrn,EO_VRD,ID,2,'VRD_Climatic_Error');
	END_IF
ELSE
	Warning:=FALSE;
END_IF

(* Execute control loop [T=500ms] *)
IF RUN AND (NOT Alarm1) THEN
	(* Calculate error *)
	Ctrl_Err:=Ctrl_SetPoint-TEMP;
	(* Init/restart operations *)
	IF NOT Ctrl_Init THEN
		Ctrl_Accel:=0;
		Ctrl_AccelTmr:=0;
		Ctrl_Err0:=Ctrl_Err;
		Ctrl_Out:=5000;
		Ctrl_Init:=TRUE;
	END_IF
	(* Calculate acceleration *)
	IF ABS(Ctrl_Err-Ctrl_Err0)>Ctrl_AccelGate OR Ctrl_AccelTmr>20 THEN
		Ctrl_Accel:=INT_TO_REAL(Ctrl_Err-Ctrl_Err0)/WORD_TO_REAL(1+Ctrl_AccelTmr);
		Ctrl_AccelTmr:=0;
		Ctrl_Err0:=Ctrl_Err;
	ELSE
		Ctrl_AccelTmr:=Ctrl_AccelTmr+1;
	END_IF
	(* Gate error *)
	IF ABS(Ctrl_Err)>Ctrl_ErrGate THEN
		(* Control loop *)
		Ctrl_Out:=Ctrl_Out+(Ctrl_Kp*Ctrl_Err)+(Ctrl_Kd*Ctrl_Accel);
	END_IF
	(* Limiter and Output *)
	Ctrl_Out:=LIMIT(0,Ctrl_Out,27000);
	OUT:=REAL_TO_WORD(Ctrl_Out);
ELSE
	Ctrl_Init:=FALSE;
	OUT:=0;
END_IF

(* Calculate position error according to feedback *)
IF ReducedRange THEN
(* SETPOINT[2..10V]-STATUS[0..10V] *)
	IF OUT<=6553 THEN Chk_Err:=0; ELSE Chk_Err:=(OUT-6553)/262; END_IF
	Chk_Err:=Chk_Err-STATUS/327;
ELSE
(* SETPOINT[0..10V]-STATUS[0..10V] *)
	Chk_Err := Chk_Err - STATUS;
END_IF

(* Check position error *)
IF ( Chk_Err<-Chk_ErrGate OR Chk_Err>Chk_ErrGate ) THEN
	IF Chk_Cnt>Chk_CntAlarm THEN
		IF NOT Alarm2 THEN
			Alarm2:=TRUE;
			LogEv(EL_Alarm,EO_VRD,ID,4,'VRD_Position_Error');
		END_IF
	ELSE
		Chk_Cnt:=Chk_Cnt+1;
	END_IF
ELSE
	Chk_Cnt:=0;
	Alarm2:=FALSE;
END_IF

(* Status temp *)
Log_AvgTemp(IN:=Temp);

Lamp.obj_Status := Status_Log;
Lamp.UpdateStatus();

(* Status color *)
   IF Alarm1 OR Alarm2 THEN Status_Log:=2; Status_Vis:=16#2020F0;
ELSIF Warning          THEN Status_Log:=1; Status_Vis:=16#20F0F0;
                       ELSE Status_Log:=0; Status_Vis:=SEL(RUN,16#006000,16#20F020);
END_IF
END_FUNCTION_BLOCK
ACTION DefaultClim:
CLIM.Points[0].X:=-300; CLIM.Points[0].Y:=400;
CLIM.Points[1].X:=-50;  CLIM.Points[1].Y:=400;
CLIM.Points[2].X:= 200; CLIM.Points[2].Y:=200;
CLIM.Points[3].X:= 300; CLIM.Points[3].Y:=200;
CLIM.Points[4].X:= 500; CLIM.Points[4].Y:=200;
CLIM.InitOK:=TRUE;
LogEv(EL_Wrn,EO_VRD,ID,1,'Climatic_Default');
END_ACTION
ACTION Init:
(* End initialization *)
InitOK:=TRUE;
END_ACTION

(* POU Plant_Objects/obj_VRD_POT, ST *)
FUNCTION_BLOCK obj_VRD_POT
(* === VALVOLA RIPARTITORE ===
   v1.0[16/04/15] - Versioning
*)
VAR_INPUT
	(* Settings *)
	ID				: BYTE;
	(* Controls *)
	RUN  			: BOOL;		(* Control input *)

	(* Physical inputs *)
	TEMP 			: INT;		(* Input temperature from sensor *)
	STATUS 			: WORD;		(* Input position from valve *)

	InitOK			: BOOL;
	Alarm1			: BOOL;
	Alarm2			: BOOL;
	Warning			: BOOL;

	Ctrl_Init		: BOOL;
	Ctrl_SetPoint	: INT;
	Ctrl_Err		: INT;			(* Current error *)
	Ctrl_Err0		: INT; 			(* Previous error *)
	Ctrl_Accel		: REAL;			(* Derivate of error *)
	Ctrl_AccelGate  : INT:=1;		(* Derivate gate *)
	Ctrl_AccelTmr	: WORD;
	Ctrl_ErrGate	: INT:=20;		(* Error gate *)
	Ctrl_Kp			: REAL:=1;		(* Proportional factor *)
	Ctrl_Kd			: REAL:=10;  	(* Derivative factor *)
	Ctrl_Out		: REAL;

	(*Chk_Err			: INT;	*)
	Chk_Err			: REAL;
	Chk_ErrGate		: INT:=50; 		(* Check error gate *)
	Chk_Cnt			: INT;
	Chk_CntAlarm	: INT:=60; 		(* Check error trigger 60s *)

	(* Status *)
	Log_AvgTemp		: AVERAGE_T;

END_VAR
VAR_IN_OUT
	CLIM		: typ_Clima;
END_VAR
VAR_OUTPUT
	(* Physical outputs *)
	OUT_CL		: BOOL;
	OUT_OP		: BOOL;

	Status_Log		: BYTE;
	Status_Vis 		: DWORD;
END_VAR
VAR
	Curve		: CHARCURVE;
	Curve_Err	: BYTE;
END_VAR
(* Check initialization *)
(*IF NOT InitOK THEN Init(); END_IF*)

(* Check max temperature *)
IF TEMP>Plant_VRD_TAlarm THEN
	IF NOT Alarm1 THEN
		Alarm1:=TRUE;
		LogEv(EL_AlarmStop,EO_VRD,ID,3,'VRD_Overtemperature');
	END_IF
END_IF

(* Check climatic setup *)
IF NOT CLIM.InitOK THEN	DefaultClim(); END_IF;
(* Calculate Setpoint *)
Curve(	IN:= T_AMB,	N:= 5, P:= CLIM.Points,			(* Given the x value as input, the corresponding y value as output is returned, if it matches the crve designed by array of points *)
		OUT=> Ctrl_SetPoint, ERR=> Curve_Err );
IF Curve_Err>0 OR Ctrl_SetPoint>Plant_VRD_TMax THEN
	Ctrl_SetPoint:=Plant_VRD_TDefault;
	IF NOT Warning THEN
		Warning:=TRUE;
		LogEv(EL_Wrn,EO_VRD,ID,2,'VRD_Climatic_Error');
	END_IF
ELSE
	Warning:=FALSE;
END_IF

(* Execute control loop [T=500ms] *)
IF RUN AND (NOT Alarm1) THEN
	(* Calculate error *)
	Ctrl_Err:=Ctrl_SetPoint-TEMP;
	(* Init/restart operations *)
	IF NOT Ctrl_Init THEN
		Ctrl_Accel:=0;
		Ctrl_AccelTmr:=0;
		Ctrl_Err0:=Ctrl_Err;
		Ctrl_Out:=0;
		Ctrl_Init:=TRUE;
	END_IF
	(* Calculate acceleration *)
	IF ABS(Ctrl_Err-Ctrl_Err0)>Ctrl_AccelGate OR Ctrl_AccelTmr>20 THEN
		Ctrl_Accel:=INT_TO_REAL(Ctrl_Err-Ctrl_Err0)/WORD_TO_REAL(1+Ctrl_AccelTmr);
		Ctrl_AccelTmr:=0;
		Ctrl_Err0:=Ctrl_Err;
	ELSE
		Ctrl_AccelTmr:=Ctrl_AccelTmr+1;
	END_IF
	(* Gate error *)
	IF ABS(Ctrl_Err)>Ctrl_ErrGate THEN
		(* Control loop *)
		Ctrl_Out:=Ctrl_Out+(Ctrl_Kp*Ctrl_Err)+(Ctrl_Kd*Ctrl_Accel);
		(* Limiter and Output *)
		Ctrl_Out:=LIMIT(0,Ctrl_Out,1000);

		(* Adjust valve position *)
		IF Ctrl_Err > 0 THEN
			OUT_CL := FALSE;
			OUT_OP :=TRUE;
		ELSE
			OUT_OP := FALSE;
			OUT_CL :=TRUE;
		END_IF
	ELSE
		OUT_OP := FALSE;
		OUT_CL := FALSE;
	END_IF

ELSE
	Ctrl_Init:=FALSE;
END_IF


(* Check position error *)

(* 0xEC00 corresponds to 0ohm, while other values are linear from 20 (10ohm -> 1%) to 2000 (1Kohm -> 100%) *)
IF Status = 16#EC00 THEN Chk_Err := Ctrl_Out;
ELSE
   Chk_Err := Ctrl_Out - Status/2;
END_IF

IF ( Chk_Err<-Chk_ErrGate OR Chk_Err>Chk_ErrGate ) THEN
	IF Chk_Cnt>Chk_CntAlarm THEN
		IF NOT Alarm2 THEN
			Alarm2:=TRUE;
			LogEv(EL_Alarm,EO_VRD,ID,4,'VRD_Position_Error');
		END_IF
	ELSE
		Chk_Cnt:=Chk_Cnt+1;
	END_IF
ELSE
	Chk_Cnt:=0;
	Alarm2:=FALSE;
END_IF

(* Status temp *)
Log_AvgTemp(IN:=Temp);
(* Status color *)
   IF Alarm1 OR Alarm2 THEN Status_Log:=2; Status_Vis:=COLOR_RED;
ELSIF Warning          THEN Status_Log:=1; Status_Vis:=COLOR_YELLOW;
                       ELSE Status_Log:=0; Status_Vis:=SEL(RUN,COLOR_LIGHT_GREEN,COLOR_GREEN);
END_IF
END_FUNCTION_BLOCK
ACTION DefaultClim:
CLIM.Points[0].X:=-300; CLIM.Points[0].Y:=400;
CLIM.Points[1].X:=-50;  CLIM.Points[1].Y:=400;
CLIM.Points[2].X:= 200; CLIM.Points[2].Y:=200;
CLIM.Points[3].X:= 300; CLIM.Points[3].Y:=200;
CLIM.Points[4].X:= 500; CLIM.Points[4].Y:=200;
CLIM.InitOK:=TRUE;
LogEv(EL_Wrn,EO_VRD,ID,1,'Climatic_Default');
END_ACTION
ACTION Init:
(* End initialization *)
Status := VRD01_ST;

InitOK:=TRUE;
END_ACTION

(* POU Plant_Objects/obj_ZTHL, ST *)
FUNCTION_BLOCK obj_ZTHL
(* === ZIGBEE AMBIENT SENSORS MT-200 ===
   v1.0[07/05/05] - Create
*)
VAR CONSTANT
	(* States *)
	WAIT_STATE			:	BYTE := 0;
	STATUS_REQUEST		:	BYTE := 1;
	LQI_REQUEST			:	BYTE := 2;
	MEAS_REQUEST		:	BYTE := 3;
	END_READ			:	BYTE := 4;
	ERROR_STATE			:	BYTE := 100;

	LQI_Threshold		:	WORD := 100;		(* Zigbee link quality minimum value *)
	LowBattVoltage		:	WORD := 270;		(* Battery is considered low when reaches 1.35V each *)
END_VAR
VAR_INPUT
	(* Settings *)
	ID				: BYTE;
	Address			: BYTE;

	Refresh_Period	: TIME:=t#5m;
	(* Controls *)
	Refresh_Auto	: BOOL:=TRUE; (* Enable automatic refresh *)
	Refresh_Now		: BOOL; 	  (* Force an immediate refresh *)

	(* Limits *)
	Tmin			: INT := 0;
	Tmax			: INT := 400;
END_VAR
VAR_IN_OUT
	(* Interface *)
	MODBUS			: obj_MODBUS_TCP;
END_VAR
VAR_OUTPUT
	OUT_TEMP		: INT;	(* Temperatura misurata [°C/10] *)
	OUT_HYGRO		: INT;	(* Umidità misurata [%] *)
	OUT_LUX			: INT;	(* Luce misurata [lux] *)
	OUT_VBATT		: INT;	(* Tensione misurata dalla batteria [V/100] *)

	OUT_LQI			: BYTE;

	NodeStatus		: WORD;
	fTemp			: BOOL;

	(* Status *)
	Status_Log		: BYTE;
	Status_Vis 		: DWORD;
END_VAR
VAR
	dly 	 		: TON := (PT:=t#5s);

	sta				: BYTE;
	retry	 		: BYTE;

	OldNodeStatus	: WORD;
	fLQI			: BOOL;
	fBatt			: BOOL;
	Quality			: FLT_EVENT;
	Battery			: FLT_EVENT;
	Temperature		: FLT_EVENT;
	Alarm			: FLT_EVENT;

	StatusOK		: BYTE;			(* 0: Status OK, >=1: Alarm and/or warning		Incremented by 1 when Alarm or Wrn occurs,
																					decremented by 1 when restored	*)
END_VAR
CASE sta OF
	WAIT_STATE: (* === Wait update signals *)
		dly(IN:=NOT (dly.Q OR Refresh_Now OR (NOT Refresh_Auto)));
		IF dly.Q OR Refresh_Now THEN
			dly.PT:=Refresh_Period;
			Refresh_Now:=FALSE;
			(*sta:=STATUS_REQUEST;*)
			sta:=LQI_REQUEST;
		END_IF

	STATUS_REQUEST:	(* Node status *)
		IF NOT (MODBUS.MB_Lock OR MODBUS.MB_Start) THEN
			MODBUS.MB_Lock:=TRUE;
			MODBUS.ID:=ID;
			MODBUS.MB_MASTER.bUNIT_ID := Address;
			MODBUS.MB_MASTER.bFUNCTION_CODE:=16#03;
			MODBUS.MB_MASTER.wREAD_ADDRESS:=16#0D;
			MODBUS.MB_MASTER.wREAD_QUANTITY:=16#1;
			MODBUS.MB_Start:=TRUE;
			sta:=LQI_REQUEST;
		END_IF

	LQI_REQUEST:	(* Link quality *)
		IF NOT MODBUS.MB_Start THEN
			IF MODBUS.MB_MASTER.wERROR<>MB_NO_ERROR THEN
				sta:=ERROR_STATE;
			ELSE
				(*NodeStatus	:=	MODBUS.MB_READBUF[0];*)

				MODBUS.ID:=ID;
				MODBUS.MB_MASTER.bUNIT_ID := Address;
				MODBUS.MB_MASTER.bFUNCTION_CODE:=16#03;
				MODBUS.MB_MASTER.wREAD_ADDRESS:=16#01;
				MODBUS.MB_MASTER.wREAD_QUANTITY:=16#1;
				MODBUS.MB_Start:=TRUE;

				sta:=MEAS_REQUEST;
			END_IF
		END_IF

	MEAS_REQUEST:	(* Measurements *)
		IF NOT MODBUS.MB_Start THEN
			IF MODBUS.MB_MASTER.wERROR<>MB_NO_ERROR THEN
				sta:=ERROR_STATE;
			ELSE

				OUT_LQI	:=	WORD_TO_BYTE(MODBUS.MB_READBUF[0]);

				MODBUS.ID:=ID;
				MODBUS.MB_MASTER.bUNIT_ID := Address;
				MODBUS.MB_MASTER.bFUNCTION_CODE:=16#03;
				MODBUS.MB_MASTER.wREAD_ADDRESS:=16#14;
				MODBUS.MB_MASTER.wREAD_QUANTITY:=16#5;
				MODBUS.MB_Start:=TRUE;

				sta:=END_READ;
			END_IF
		END_IF

	END_READ:	IF NOT MODBUS.MB_Start THEN
			IF MODBUS.MB_MASTER.wERROR<>MB_NO_ERROR THEN
				sta:=ERROR_STATE;
			ELSE
				OUT_TEMP	:=	WORD_TO_INT(MODBUS.MB_READBUF[0]);
				OUT_HYGRO	:=	WORD_TO_INT(MODBUS.MB_READBUF[1]);
				OUT_LUX		:=	WORD_TO_INT(MODBUS.MB_READBUF[2]);
				OUT_VBATT	:=	WORD_TO_INT(MODBUS.MB_READBUF[3]);
				sta:=WAIT_STATE;
				MODBUS.MB_Lock:=FALSE;
			END_IF
		END_IF

	ERROR_STATE:
			MODBUS.MB_Lock:=FALSE;
			(* Retries *)
			retry:=retry+1;
			IF retry>3 THEN
				retry:=0;
				IF Status_Log<>2 THEN
					LogEv(EL_Alarm,EO_ZTHL,ID,4,'');
				END_IF
				Status_Log:=2;
				Status_Vis:=COLOR_RED;
			END_IF
			sta:=WAIT_STATE;

ELSE
			sta:=WAIT_STATE;
END_CASE

(* Check Status *)
(*
IF NodeStatus <> OldNodeStatus THEN
	IF NodeStatus = 3 THEN
		LogEv(EL_Alarm,EO_ZTHL,ID,3,'');
		Status_Log:=2;
	ELSE
		Status_Log:=0;
	END_IF

	OldNodeStatus := NodeStatus;
END_IF*)

(* Check Link quality *)
IF OUT_LQI > LQI_Threshold THEN fLQI := TRUE;
ELSE fLQI := FALSE;
END_IF

Quality(IN:=fLQI);

IF Quality.EVL THEN
	LogEv(SEL(OUT_LQI<>0,EL_Alarm,EL_Wrn),EO_ZTHL,ID,SEL(OUT_LQI<>0,7,2),WORD_TO_STRING(OUT_LQI));
	Status_Log := SEL(OUT_LQI<>0,2,1);
	StatusOK := StatusOK + 1;
END_IF

IF Quality.EVH THEN StatusOK := SEL(StatusOK=0, StatusOK-1, 0); END_IF

(* If probe (node) is present proceed checking other warnings, otherwise don't transmit anything *)
IF OUT_LQI <> 0 THEN

	(* Check battery voltage *)
	IF OUT_VBATT < LowBattVoltage THEN fBatt := TRUE;
	ELSE fBatt := FALSE;
	END_IF
	
	Battery(IN:=fBatt);
	
	IF Battery.EVH THEN
		LogEv(EL_Wrn,EO_ZTHL,ID,6,'');
		StatusOK := StatusOK + 1;
	END_IF

	IF Battery.EVL THEN StatusOK := SEL(StatusOK=0, StatusOK-1, 0); END_IF

	(* Check Node temperature *)
	IF OUT_TEMP < Tmin OR OUT_TEMP > Tmax THEN
		fTemp := TRUE;
	ELSE
		fTemp := FALSE;
	END_IF

	Temperature(IN:=fTemp);

	IF Temperature.EVH THEN
		LogEv(EL_Wrn,EO_ZTHL,ID,5,INT_TO_STRING(OUT_TEMP));
		Status_Log := 1;
		StatusOK := StatusOK + 1;
	END_IF

	IF Temperature.EVL THEN StatusOK := SEL(StatusOK=0, StatusOK-1, 0); END_IF

END_IF

Alarm(IN:=(StatusOK=0));

IF Alarm.EVH THEN
	Status_Log := 0;
	LogEv(EL_Log,EO_ZTHL,ID,1,'');
END_IF

IF Status_Log = 2 THEN Status_Vis := COLOR_RED;
ELSIF Status_Log = 1 THEN Status_Vis := COLOR_YELLOW;
ELSE Status_Vis := COLOR_GREEN;
END_IF
END_FUNCTION_BLOCK
ACTION AddLogData:
Logger.s1:=INSERT('&ZTHL=',BYTE_TO_STRING(ID),4);
IF ID<10 THEN Logger.s1:=INSERT(Logger.s1,'0',4); END_IF

Logger.s1:=CONCAT(Logger.s1,BYTE_TO_STRING(OUT_LQI));			Logger.s1:=CONCAT(Logger.s1,';');
Logger.s1:=CONCAT(Logger.s1,INT_TO_STRING(OUT_TEMP ));			Logger.s1:=CONCAT(Logger.s1,';');
Logger.s1:=CONCAT(Logger.s1,INT_TO_STRING(OUT_HYGRO ));			Logger.s1:=CONCAT(Logger.s1,';');
Logger.s1:=CONCAT(Logger.s1,INT_TO_STRING(OUT_LUX));			Logger.s1:=CONCAT(Logger.s1,';');
Logger.s1:=CONCAT(Logger.s1,INT_TO_STRING(OUT_VBATT));			Logger.s1:=CONCAT(Logger.s1,';');

Logger.s1:=CONCAT(Logger.s1,BYTE_TO_STRING(Status_Log));
ADDSTRING(ADR(Logger.TData), ADR(Logger.s1), Logger.TLen);
END_ACTION

(* POU Utils Functions/PLANT_STATUS, ST *)
FUNCTION_BLOCK PLANT_STATUS
VAR_INPUT
	obj_Status		:	WORD;
END_VAR
VAR_OUTPUT
END_VAR
VAR
	PLANT_STATUS	:	WORD;

	Pwm				:	TON := (PT:=T#1s);
END_VAR
CASE plant_Status OF

	0:	(* Plant OK - Everything works well *)
		Pwm(IN:=FALSE);							(* Stop timer if running *)
		LAMP_AL := FALSE;						(* Keep the lamp switched off *)

	1:	(* Plant in warning *)
		Pwm(IN:= NOT(Pwm.Q));

		IF Pwm.Q THEN
			LAMP_AL := NOT LAMP_AL;				(* Toggle output *)
		END_IF

	2:	(* Plant in alarm *)
		Pwm(IN:=FALSE);							(* Stop timer if running *)
		LAMP_AL	:= TRUE;						(* Keep the lamp switched on *)

END_CASE

plant_Status := 0;		(* Reset plant status *)
END_FUNCTION_BLOCK
ACTION UpdateStatus:
IF plant_Status = 2 THEN

	RETURN;					(* If plant already in alarm condition do nothing *)

ELSE

		IF obj_Status <> 0 THEN
			plant_Status := obj_Status;			(* If plant in warning/normal condition and current object in alarm, update plant status *)
		END_IF
END_IF
END_ACTION

(* POU PLC_WDT, ST *)
FUNCTION PLC_WDT: DWORD VAR_INPUT dwEvent: DWORD; dwFilter: DWORD; dwOwner: DWORD; END_VAR
LogEv(EL_AlarmStop,EO_SYS,1,10,'Watchdog');
END_FUNCTION

(* POU Utils Functions/RAW16TOHEXSTR, ST *)
FUNCTION RAW16TOHEXSTR : STRING(128)
VAR_INPUT
	pData: POINTER TO BYTE;
	DataLen: BYTE;
END_VAR
VAR
	pt: POINTER TO BYTE;
	xl: BYTE;
END_VAR
pt:=ADR(RAW16TOHEXSTR);
xl:=0;

WHILE DataLen>0 AND xl<120 DO

	pData:=pData+1;

	pt^ := (pData^ / 16#10) + 48 + (((pData^ / 16#10)/10)*7);
	pt:=pt+1;
	pt^ := (pData^ AND 16#0F)  + 48 + (((pData^ AND 16#0F)/10)*7);
	pt:=pt+1;

	pData:=pData-1;

	pt^ := (pData^ / 16#10) + 48 + (((pData^ / 16#10)/10)*7);
	pt:=pt+1;
	pt^ := (pData^ AND 16#0F)  + 48 + (((pData^ AND 16#0F)/10)*7);
	pt:=pt+1;

	xl:=xl+4;

	DataLen:=DataLen-2;
	pData:=pData+2;

END_WHILE

pt^:=0;
END_FUNCTION

(* POU Utils/RTC_Update, ST *)
FUNCTION RTC_Update : BOOL
VAR
	T: DT;
	TS: STRING;
	TS2: STRING;
	Hour: BYTE;
	Minute: BYTE;
END_VAR
(* Get RTC time *)
T:=SysRtcGetTime(TRUE);
Sys.Time_CT_DT:=T;
(* Calculate variables *)
TS:=DT_TO_STRING(T);
Sys.Time_LogString:=DELETE(STR:=TS, LEN:=3, POS:=1);
TS2:=MID(STR:=TS, LEN:=4, POS:= 4); Sys.Time_Year 	:=STRING_TO_WORD(TS2);
TS2:=MID(STR:=TS, LEN:=2, POS:= 9); Sys.Time_Month	:=STRING_TO_BYTE(TS2);
TS2:=MID(STR:=TS, LEN:=2, POS:=12); Sys.Time_Day  	:=STRING_TO_BYTE(TS2);
Sys.Time_CT_Day:=(32*(Sys.Time_Month-1)+Sys.Time_Day-1);
TS2:=MID(STR:=TS, LEN:=2, POS:=15); Hour			:=STRING_TO_BYTE(TS2);
TS2:=MID(STR:=TS, LEN:=2, POS:=18); Minute		 	:=STRING_TO_BYTE(TS2);
Sys.Time_CT_Quarter:=Hour*4+(Minute/15);
END_FUNCTION

(* POU Utils Functions/SHIFT_ARRAY, ST *)
FUNCTION SHIFT_ARRAY : BOOL
VAR_INPUT
	pData	:	POINTER TO ARRAY [1..2] OF WORD;
	Size	:	BYTE;
END_VAR
VAR
	pNew	:	POINTER TO WORD;
	i		:	BYTE;
END_VAR
(* Shift right *)
FOR i:=1 TO (Size-1) BY 1 DO

	(*pNew := pData + 1;*)
	pData^[i] := pData^[i+1];
	(*pData := pData + 1;*)

END_FOR
END_FUNCTION

(* Visualisation PLC_VISU
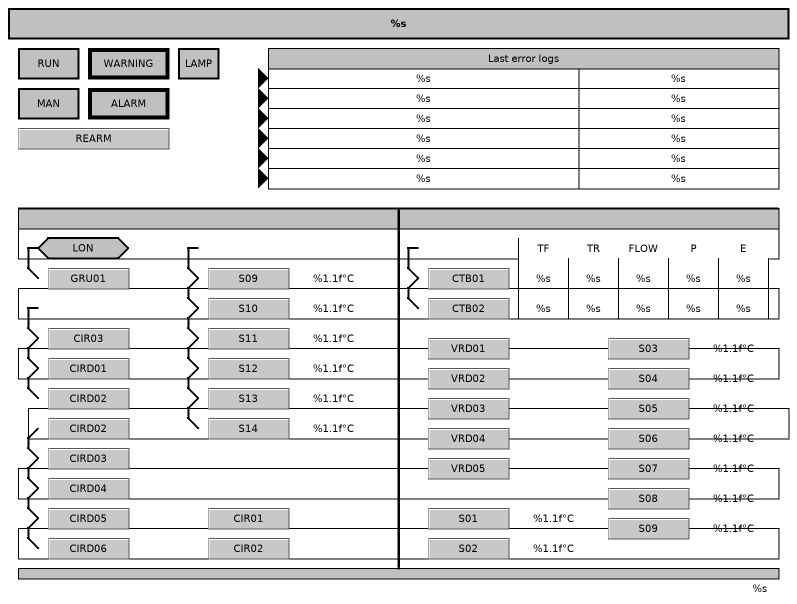
rectangle at (10,10)-(791,41): text "%s"; shows .Plant_NAME
rectangle at (530,580)-(771,601): text "%s"; shows Sys.Time_LogString
rounded rectangle at (20,50)-(81,81): text "RUN"; alarm colour if NOT Mode_Manual; runs INTERN ASSIGN Mode_Manual:=(FALSE)
rounded rectangle at (20,90)-(81,121): text "MAN"; alarm colour if Mode_Manual; runs INTERN ASSIGN Mode_Manual:=(TRUE)
rectangle at (580,70)-(781,91): text "%s"; shows Sys.LastLogs_Msg[0]
polygon at (260,170)-(270,190): invisible if Sys.LastLogs_Idx<>0
rectangle at (580,90)-(781,111): text "%s"; shows Sys.LastLogs_Msg[1]
polygon at (260,70)-(270,90): invisible if Sys.LastLogs_Idx<>1
rectangle at (580,110)-(781,131): text "%s"; shows Sys.LastLogs_Msg[2]
polygon at (260,90)-(270,110): invisible if Sys.LastLogs_Idx<>2
rectangle at (580,130)-(781,151): text "%s"; shows Sys.LastLogs_Msg[3]
polygon at (260,110)-(270,130): invisible if Sys.LastLogs_Idx<>3
rectangle at (580,150)-(781,171): text "%s"; shows Sys.LastLogs_Msg[4]
polygon at (260,130)-(270,150): invisible if Sys.LastLogs_Idx<>4
rectangle at (580,170)-(781,191): text "%s"; shows Sys.LastLogs_Msg[5]
polygon at (260,150)-(270,170): invisible if Sys.LastLogs_Idx<>5
rectangle at (270,70)-(581,91): text "%s"; shows Sys.LastLogs_Dat[0]
rectangle at (270,90)-(581,111): text "%s"; shows Sys.LastLogs_Dat[1]
rectangle at (270,110)-(581,131): text "%s"; shows Sys.LastLogs_Dat[2]
rectangle at (270,130)-(581,151): text "%s"; shows Sys.LastLogs_Dat[3]
rectangle at (270,150)-(581,171): text "%s"; shows Sys.LastLogs_Dat[4]
rectangle at (270,170)-(581,191): text "%s"; shows Sys.LastLogs_Dat[5]
rectangle at (90,90)-(171,121): text "ALARM"; alarm colour if Sys.Alarm; runs INTERN ASSIGN Mode_Manual:=(FALSE)
rectangle at (90,50)-(171,81): text "WARNING"; alarm colour if Sys.Warning; runs INTERN ASSIGN Mode_Manual:=(TRUE)
button at (20,130)-(171,151): text "REARM"; runs INTERN ASSIGN Sys.Alarm:=(FALSE);INTERN ASSIGN Sys.Warning:=(FALSE)
button at (430,270)-(511,291): text "CTB01"
rectangle at (270,50)-(781,71): text "Last error logs"
rectangle at (520,240)-(571,261): text "TF"
rectangle at (620,240)-(671,261): text "FLOW"
rectangle at (670,240)-(721,261): text "P"
rectangle at (720,240)-(771,261): text "E"
rectangle at (570,240)-(621,261): text "TR"
rectangle at (520,270)-(571,291): text "%s"; shows .CTB01.M1.utFTemp.Value
rectangle at (620,270)-(671,291): text "%s"; shows .CTB01.M1.utFlow.Value
rectangle at (670,270)-(721,291): text "%s"; shows CTB01.M1.utPower.Value
rectangle at (720,270)-(771,291): text "%s"; shows CTB01.M1.utEnergy.Value
rectangle at (570,270)-(621,291): text "%s"; shows .CTB01.M1.utRTemp.Value
button at (50,390)-(131,411): text "CIRD02"
button at (50,420)-(131,441): text "CIRD02"
button at (50,450)-(131,471): text "CIRD03"
button at (50,330)-(131,351): text "CIR03"
button at (50,480)-(131,501): text "CIRD04"
button at (50,360)-(131,381): text "CIRD01"
button at (430,510)-(511,531): text "S01"; opens Vis_VRD02
button at (430,540)-(511,561): text "S02"; opens Vis_VRD02
button at (610,340)-(691,361): text "S03"; opens Vis_VRD02
button at (210,270)-(291,291): text "S09"; opens Vis_VRD02
button at (210,300)-(291,321): text "S10"; opens Vis_VRD02
button at (210,330)-(291,351): text "S11"; opens Vis_VRD02
button at (210,360)-(291,381): text "S12"; opens Vis_VRD02
button at (210,390)-(291,411): text "S13"; opens Vis_VRD02
button at (210,420)-(291,441): text "S14"; opens Vis_VRD02
rectangle at (510,510)-(601,531): text "%1.1f°C"; shows INT_TO_REAL(.TPV01.IN)/10
rectangle at (510,540)-(601,561): text "%1.1f°C"; shows INT_TO_REAL(.TPV02.IN)/10
rectangle at (690,340)-(781,361): text "%1.1f°C"; shows INT_TO_REAL(.TPV03.IN)/10
rectangle at (290,270)-(381,291): text "%1.1f°C"; shows INT_TO_REAL(ZTHL09.OUT_TEMP)/10
rectangle at (290,300)-(381,321): text "%1.1f°C"; shows INT_TO_REAL(ZTHL10.OUT_TEMP)/10
rectangle at (290,330)-(381,351): text "%1.1f°C"; shows INT_TO_REAL(.ZTHL11.OUT_TEMP)/10
rectangle at (290,360)-(381,381): text "%1.1f°C"; shows INT_TO_REAL(ZTHL12.OUT_TEMP)/10
rectangle at (290,390)-(381,411): text "%1.1f°C"; shows INT_TO_REAL(ZTHL13.OUT_TEMP)/10
rectangle at (290,420)-(381,441): text "%1.1f°C"; shows INT_TO_REAL(ZTHL14.OUT_TEMP)/10
polygon at (40,240)-(130,260): text "LON"
button at (50,270)-(131,291): text "GRU01"; opens Vis_CAL01
button at (50,510)-(131,531): text "CIRD05"
button at (50,540)-(131,561): text "CIRD06"
button at (430,340)-(511,361): text "VRD01"; opens Vis_VRD02
button at (430,370)-(511,391): text "VRD02"; opens Vis_VRD02
rounded rectangle at (180,50)-(221,81): text "LAMP"; alarm colour if LAMP_AL
button at (610,370)-(691,391): text "S04"; opens Vis_VRD02
button at (610,400)-(691,421): text "S05"; opens Vis_VRD02
button at (610,430)-(691,451): text "S06"; opens Vis_VRD02
rectangle at (690,370)-(781,391): text "%1.1f°C"; shows INT_TO_REAL(.TPV04.IN)/10
rectangle at (690,400)-(781,421): text "%1.1f°C"; shows INT_TO_REAL(.TPV05.IN)/10
rectangle at (690,430)-(781,451): text "%1.1f°C"; shows INT_TO_REAL(.TPV06.IN)/10
button at (610,460)-(691,481): text "S07"; opens Vis_VRD02
button at (610,490)-(691,511): text "S08"; opens Vis_VRD02
button at (610,520)-(691,541): text "S09"; opens Vis_VRD02
rectangle at (690,460)-(781,481): text "%1.1f°C"; shows INT_TO_REAL(.TPV07.IN)/10
rectangle at (690,490)-(781,511): text "%1.1f°C"; shows INT_TO_REAL(.TPV08.IN)/10
rectangle at (690,520)-(781,541): text "%1.1f°C"; shows INT_TO_REAL(.TPV09.IN)/10
button at (430,400)-(511,421): text "VRD03"; opens Vis_VRD02
button at (430,430)-(511,451): text "VRD04"; opens Vis_VRD02
button at (430,460)-(511,481): text "VRD05"; opens Vis_VRD02
button at (210,510)-(291,531): text "CIR01"; opens Vis_VRD02
button at (210,540)-(291,561): text "CIR02"; opens Vis_VRD02
button at (430,300)-(511,321): text "CTB02"
rectangle at (520,300)-(571,321): text "%s"; shows .CTB02.M1.utFTemp.Value
rectangle at (570,300)-(621,321): text "%s"; shows .CTB02.M1.utRTemp.Value
rectangle at (620,300)-(671,321): text "%s"; shows .CTB02.M1.utFlow.Value
rectangle at (670,300)-(721,321): text "%s"; shows CTB02.M1.utPower.Value
rectangle at (720,300)-(771,321): text "%s"; shows CTB02.M1.utEnergy.Value
32 more shapes without text or variables
36 elements of other kinds (tables, trends, ...) not read
*)

